Yaskawa INFORM job: A_NAIHAN_0617_1_PAINT_2.JBI

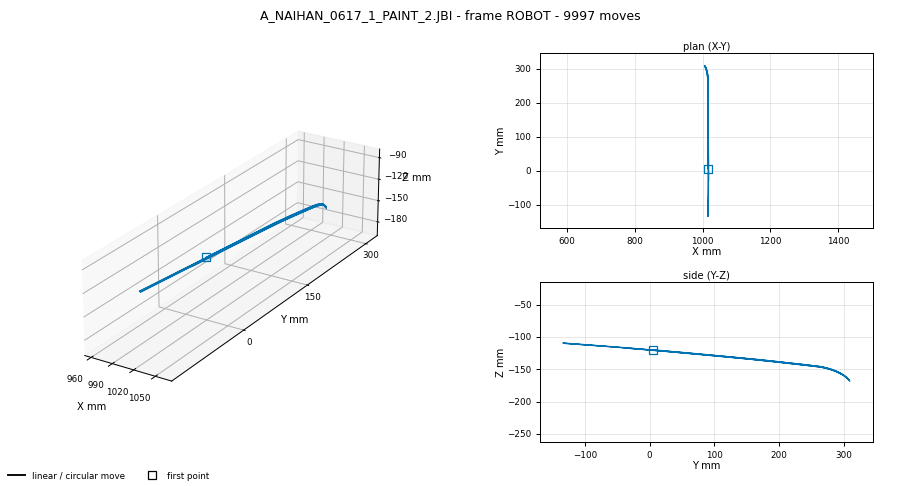
[picture p0: tool path of A_NAIHAN_0617_1_PAINT_2.JBI in frame ROBOT, 9997 of 9997 moves have a stored position in this frame; points joined in program order, loops and branches not executed]
/JOB
//NAME A_NAIHAN_0617_1_PAINT2
//POS
///NPOS 9997,0,0,0,0,0
///TOOL 1
///USER 0
///POSTYPE ROBOT
///RECTAN
///RCONF 0,0,0,0,1,0,0,0,0,0,0,0,0,0,0,0,0,0,0,0,0,0,0,0
C00000=1015.956,5.375,-119.573,-24.182,21.519,-42.790
C00001=1015.955,5.769,-119.606,-24.182,21.518,-42.785
C00002=1015.954,6.162,-119.640,-24.183,21.519,-42.779
C00003=1015.954,6.555,-119.673,-24.184,21.517,-42.775
C00004=1015.952,6.948,-119.706,-24.185,21.517,-42.770
C00005=1015.951,7.339,-119.740,-24.185,21.517,-42.764
C00006=1015.951,7.726,-119.773,-24.186,21.516,-42.761
C00007=1015.950,8.110,-119.806,-24.187,21.516,-42.755
C00008=1015.949,8.491,-119.838,-24.187,21.515,-42.751
C00009=1015.948,8.869,-119.869,-24.188,21.515,-42.746
C00010=1015.947,9.245,-119.902,-24.189,21.514,-42.740
C00011=1015.945,9.621,-119.935,-24.189,21.514,-42.737
C00012=1015.945,9.998,-119.966,-24.190,21.513,-42.731
C00013=1015.944,10.376,-119.999,-24.191,21.513,-42.726
C00014=1015.943,10.757,-120.031,-24.191,21.513,-42.722
C00015=1015.942,11.139,-120.064,-24.192,21.512,-42.716
C00016=1015.940,11.526,-120.098,-24.192,21.511,-42.713
C00017=1015.940,11.912,-120.131,-24.193,21.512,-42.707
C00018=1015.938,12.298,-120.164,-24.193,21.510,-42.703
C00019=1015.938,12.685,-120.197,-24.194,21.510,-42.698
C00020=1015.936,13.071,-120.230,-24.195,21.511,-42.693
C00021=1015.935,13.458,-120.263,-24.196,21.509,-42.689
C00022=1015.933,13.845,-120.297,-24.196,21.509,-42.683
C00023=1015.933,14.233,-120.330,-24.197,21.509,-42.680
C00024=1015.931,14.621,-120.363,-24.198,21.508,-42.674
C00025=1015.930,15.011,-120.397,-24.198,21.508,-42.670
C00026=1015.928,15.400,-120.430,-24.199,21.507,-42.665
C00027=1015.927,15.790,-120.464,-24.200,21.507,-42.659
C00028=1015.927,16.181,-120.498,-24.200,21.506,-42.656
C00029=1015.925,16.573,-120.531,-24.201,21.506,-42.650
C00030=1015.923,16.965,-120.565,-24.201,21.505,-42.646
C00031=1015.922,17.359,-120.599,-24.202,21.505,-42.641
C00032=1015.921,17.753,-120.633,-24.203,21.505,-42.635
C00033=1015.920,18.148,-120.667,-24.203,21.504,-42.632
C00034=1015.917,18.544,-120.701,-24.204,21.503,-42.626
C00035=1015.917,18.940,-120.736,-24.205,21.503,-42.622
C00036=1015.915,19.338,-120.770,-24.205,21.503,-42.617
C00037=1015.914,19.548,-120.788,-24.206,21.503,-42.613
C00038=1015.913,19.785,-120.809,-24.206,21.502,-42.610
C00039=1015.912,20.051,-120.831,-24.207,21.503,-42.606
C00040=1015.912,20.337,-120.857,-24.207,21.501,-42.604
C00041=1015.910,20.635,-120.882,-24.207,21.501,-42.602
C00042=1015.909,20.926,-120.907,-24.208,21.502,-42.599
C00043=1015.908,21.198,-120.931,-24.208,21.501,-42.597
C00044=1015.907,21.443,-120.952,-24.209,21.501,-42.593
C00045=1015.905,21.856,-120.988,-24.210,21.501,-42.586
C00046=1015.904,22.231,-121.020,-24.210,21.500,-42.584
C00047=1015.902,22.553,-121.049,-24.211,21.500,-42.580
C00048=1015.901,22.819,-121.071,-24.211,21.500,-42.577
C00049=1015.900,23.051,-121.092,-24.211,21.499,-42.573
C00050=1015.899,23.286,-121.112,-24.212,21.498,-42.567
C00051=1015.898,23.557,-121.136,-24.213,21.498,-42.564
C00052=1015.897,23.888,-121.165,-24.213,21.498,-42.562
C00053=1015.895,24.271,-121.198,-24.213,21.497,-42.558
C00054=1015.893,24.669,-121.233,-24.214,21.497,-42.553
C00055=1015.891,25.069,-121.267,-24.215,21.497,-42.549
C00056=1015.890,25.468,-121.302,-24.215,21.496,-42.543
C00057=1015.888,25.868,-121.337,-24.216,21.496,-42.540
C00058=1015.886,26.267,-121.372,-24.217,21.496,-42.534
C00059=1015.884,26.666,-121.407,-24.218,21.495,-42.529
C00060=1015.882,27.066,-121.441,-24.218,21.494,-42.525
C00061=1015.881,27.465,-121.476,-24.219,21.495,-42.520
C00062=1015.879,27.865,-121.511,-24.219,21.493,-42.516
C00063=1015.877,28.264,-121.545,-24.220,21.493,-42.510
C00064=1015.875,28.664,-121.581,-24.221,21.493,-42.507
C00065=1015.873,29.063,-121.616,-24.221,21.492,-42.501
C00066=1015.872,29.462,-121.651,-24.222,21.492,-42.497
C00067=1015.869,29.863,-121.686,-24.223,21.492,-42.492
C00068=1015.867,30.262,-121.720,-24.223,21.491,-42.488
C00069=1015.865,30.661,-121.756,-24.224,21.491,-42.483
C00070=1015.863,31.061,-121.790,-24.224,21.490,-42.479
C00071=1015.861,31.461,-121.826,-24.225,21.490,-42.474
C00072=1015.859,31.860,-121.861,-24.226,21.489,-42.469
C00073=1015.857,32.260,-121.895,-24.226,21.489,-42.464
C00074=1015.855,32.659,-121.930,-24.227,21.489,-42.461
C00075=1015.853,33.059,-121.966,-24.228,21.489,-42.455
C00076=1015.850,33.459,-122.001,-24.228,21.487,-42.451
C00077=1015.849,33.858,-122.036,-24.229,21.488,-42.446
C00078=1015.846,34.258,-122.071,-24.229,21.487,-42.442
C00079=1015.844,34.658,-122.106,-24.230,21.486,-42.437
C00080=1015.841,35.057,-122.142,-24.231,21.486,-42.433
C00081=1015.840,35.457,-122.176,-24.231,21.486,-42.428
C00082=1015.837,35.857,-122.211,-24.232,21.486,-42.424
C00083=1015.835,36.256,-122.247,-24.233,21.485,-42.418
C00084=1015.832,36.656,-122.282,-24.233,21.484,-42.414
C00085=1015.830,37.057,-122.317,-24.234,21.485,-42.409
C00086=1015.828,37.456,-122.353,-24.235,21.484,-42.405
C00087=1015.825,37.856,-122.388,-24.235,21.483,-42.400
C00088=1015.823,38.256,-122.423,-24.236,21.483,-42.396
C00089=1015.821,38.655,-122.459,-24.237,21.483,-42.391
C00090=1015.818,39.056,-122.494,-24.237,21.483,-42.387
C00091=1015.816,39.455,-122.529,-24.238,21.482,-42.383
C00092=1015.813,39.855,-122.565,-24.238,21.481,-42.378
C00093=1015.811,40.256,-122.600,-24.239,21.481,-42.374
C00094=1015.809,40.655,-122.635,-24.240,21.481,-42.369
C00095=1015.806,41.055,-122.670,-24.240,21.481,-42.365
C00096=1015.804,41.455,-122.706,-24.241,21.480,-42.359
C00097=1015.801,41.855,-122.742,-24.241,21.479,-42.356
C00098=1015.798,42.255,-122.777,-24.242,21.479,-42.352
C00099=1015.796,42.654,-122.812,-24.243,21.479,-42.347
C00100=1015.794,43.055,-122.847,-24.243,21.479,-42.343
C00101=1015.791,43.455,-122.884,-24.244,21.479,-42.338
C00102=1015.788,43.855,-122.918,-24.244,21.477,-42.333
C00103=1015.786,44.255,-122.954,-24.245,21.477,-42.330
C00104=1015.783,44.655,-122.990,-24.246,21.477,-42.325
C00105=1015.780,45.055,-123.025,-24.246,21.477,-42.321
C00106=1015.778,45.455,-123.061,-24.247,21.477,-42.316
C00107=1015.775,45.855,-123.096,-24.247,21.475,-42.311
C00108=1015.772,46.255,-123.132,-24.248,21.475,-42.308
C00109=1015.770,46.655,-123.168,-24.249,21.475,-42.302
C00110=1015.766,47.055,-123.203,-24.249,21.475,-42.299
C00111=1015.764,47.455,-123.239,-24.250,21.474,-42.295
C00112=1015.761,47.855,-123.274,-24.251,21.474,-42.290
C00113=1015.758,48.256,-123.311,-24.251,21.474,-42.286
C00114=1015.756,48.656,-123.345,-24.251,21.472,-42.282
C00115=1015.753,49.056,-123.381,-24.252,21.473,-42.277
C00116=1015.750,49.455,-123.417,-24.253,21.472,-42.273
C00117=1015.747,49.856,-123.452,-24.254,21.472,-42.268
C00118=1015.744,50.256,-123.489,-24.254,21.472,-42.264
C00119=1015.740,50.656,-123.524,-24.255,21.471,-42.260
C00120=1015.739,51.056,-123.560,-24.255,21.471,-42.255
C00121=1015.735,51.457,-123.595,-24.256,21.471,-42.251
C00122=1015.732,51.857,-123.631,-24.256,21.470,-42.247
C00123=1015.729,52.257,-123.667,-24.257,21.469,-42.243
C00124=1015.726,52.657,-123.703,-24.258,21.469,-42.238
C00125=1015.723,53.057,-123.739,-24.258,21.469,-42.234
C00126=1015.719,53.457,-123.774,-24.259,21.468,-42.230
C00127=1015.717,53.857,-123.810,-24.259,21.468,-42.225
C00128=1015.714,54.257,-123.846,-24.260,21.468,-42.221
C00129=1015.711,54.658,-123.882,-24.260,21.468,-42.218
C00130=1015.708,55.058,-123.918,-24.261,21.468,-42.212
C00131=1015.705,55.458,-123.953,-24.262,21.467,-42.209
C00132=1015.702,55.858,-123.989,-24.262,21.467,-42.205
C00133=1015.698,56.258,-124.026,-24.263,21.465,-42.201
C00134=1015.695,56.659,-124.062,-24.264,21.466,-42.196
C00135=1015.691,57.059,-124.098,-24.264,21.465,-42.192
C00136=1015.688,57.459,-124.133,-24.264,21.465,-42.188
C00137=1015.685,57.859,-124.169,-24.265,21.465,-42.183
C00138=1015.682,58.259,-124.205,-24.266,21.464,-42.179
C00139=1015.679,58.659,-124.241,-24.266,21.464,-42.175
C00140=1015.675,59.059,-124.277,-24.267,21.463,-42.172
C00141=1015.671,59.460,-124.313,-24.268,21.464,-42.166
C00142=1015.668,59.860,-124.349,-24.268,21.463,-42.163
C00143=1015.665,60.260,-124.385,-24.269,21.463,-42.159
C00144=1015.661,60.660,-124.421,-24.269,21.462,-42.155
C00145=1015.658,61.060,-124.457,-24.270,21.462,-42.150
C00146=1015.655,61.460,-124.493,-24.270,21.462,-42.146
C00147=1015.651,61.861,-124.529,-24.271,21.461,-42.142
C00148=1015.648,62.261,-124.565,-24.271,21.461,-42.139
C00149=1015.644,62.681,-124.603,-24.272,21.460,-42.133
C00150=1015.642,62.934,-124.626,-24.272,21.460,-42.131
C00151=1015.640,63.201,-124.650,-24.273,21.460,-42.129
C00152=1015.638,63.450,-124.673,-24.273,21.459,-42.127
C00153=1015.636,63.668,-124.693,-24.274,21.460,-42.124
C00154=1015.634,63.875,-124.711,-24.274,21.460,-42.122
C00155=1015.631,64.093,-124.730,-24.274,21.459,-42.120
C00156=1015.629,64.322,-124.751,-24.274,21.459,-42.116
C00157=1015.627,64.558,-124.773,-24.275,21.459,-42.115
C00158=1015.625,64.794,-124.794,-24.275,21.458,-42.113
C00159=1015.623,65.024,-124.815,-24.275,21.458,-42.111
C00160=1015.621,65.245,-124.835,-24.276,21.459,-42.108
C00161=1015.619,65.458,-124.853,-24.276,21.458,-42.106
C00162=1015.616,65.866,-124.891,-24.277,21.458,-42.102
C00163=1015.611,66.264,-124.927,-24.277,21.457,-42.098
C00164=1015.609,66.665,-124.963,-24.278,21.457,-42.094
C00165=1015.604,67.067,-124.999,-24.278,21.457,-42.089
C00166=1015.600,67.470,-125.036,-24.279,21.457,-42.085
C00167=1015.597,67.875,-125.072,-24.279,21.456,-42.082
C00168=1015.593,68.281,-125.110,-24.280,21.456,-42.078
C00169=1015.590,68.689,-125.146,-24.280,21.455,-42.074
C00170=1015.586,69.097,-125.183,-24.281,21.455,-42.069
C00171=1015.581,69.507,-125.221,-24.282,21.455,-42.065
C00172=1015.577,69.918,-125.258,-24.282,21.454,-42.061
C00173=1015.573,70.330,-125.295,-24.283,21.454,-42.058
C00174=1015.570,70.741,-125.332,-24.283,21.453,-42.054
C00175=1015.566,71.152,-125.369,-24.284,21.454,-42.049
C00176=1015.562,71.563,-125.406,-24.285,21.453,-42.045
C00177=1015.557,71.975,-125.444,-24.285,21.453,-42.041
C00178=1015.553,72.388,-125.482,-24.285,21.452,-42.037
C00179=1015.550,72.804,-125.520,-24.286,21.452,-42.034
C00180=1015.545,73.221,-125.557,-24.287,21.452,-42.028
C00181=1015.541,73.641,-125.596,-24.287,21.452,-42.025
C00182=1015.539,73.853,-125.615,-24.288,21.451,-42.023
C00183=1015.537,74.065,-125.634,-24.288,21.451,-42.021
C00184=1015.535,74.278,-125.653,-24.288,21.451,-42.019
C00185=1015.532,74.490,-125.673,-24.288,21.451,-42.017
C00186=1015.530,74.704,-125.692,-24.289,21.450,-42.015
C00187=1015.528,74.918,-125.712,-24.289,21.451,-42.012
C00188=1015.526,75.131,-125.731,-24.289,21.451,-42.010
C00189=1015.523,75.344,-125.751,-24.290,21.450,-42.008
C00190=1015.519,75.763,-125.789,-24.290,21.450,-42.004
C00191=1015.514,76.175,-125.826,-24.291,21.449,-42.001
C00192=1015.511,76.577,-125.862,-24.291,21.449,-41.997
C00193=1015.507,76.972,-125.898,-24.292,21.449,-41.994
C00194=1015.503,77.360,-125.934,-24.292,21.448,-41.989
C00195=1015.498,77.746,-125.969,-24.293,21.447,-41.986
C00196=1015.495,78.133,-126.005,-24.293,21.448,-41.980
C00197=1015.490,78.523,-126.040,-24.294,21.447,-41.977
C00198=1015.485,78.920,-126.076,-24.294,21.447,-41.973
C00199=1015.481,79.326,-126.113,-24.295,21.447,-41.970
C00200=1015.477,79.740,-126.152,-24.296,21.447,-41.966
C00201=1015.475,79.950,-126.170,-24.296,21.446,-41.964
C00202=1015.473,80.162,-126.190,-24.296,21.446,-41.962
C00203=1015.471,80.375,-126.209,-24.296,21.446,-41.960
C00204=1015.468,80.588,-126.228,-24.297,21.446,-41.958
C00205=1015.466,80.800,-126.247,-24.297,21.445,-41.956
C00206=1015.463,81.013,-126.267,-24.297,21.445,-41.955
C00207=1015.461,81.225,-126.287,-24.297,21.445,-41.953
C00208=1015.459,81.437,-126.306,-24.298,21.445,-41.951
C00209=1015.456,81.650,-126.326,-24.298,21.445,-41.949
C00210=1015.453,81.862,-126.345,-24.298,21.444,-41.947
C00211=1015.451,82.073,-126.364,-24.299,21.445,-41.944
C00212=1015.449,82.284,-126.384,-24.299,21.444,-41.942
C00213=1015.444,82.705,-126.422,-24.299,21.444,-41.938
C00214=1015.440,83.126,-126.460,-24.300,21.444,-41.935
C00215=1015.434,83.545,-126.499,-24.300,21.444,-41.931
C00216=1015.430,83.962,-126.537,-24.301,21.443,-41.927
C00217=1015.425,84.378,-126.575,-24.301,21.443,-41.923
C00218=1015.420,84.792,-126.613,-24.302,21.443,-41.920
C00219=1015.416,85.204,-126.651,-24.302,21.442,-41.916
C00220=1015.411,85.615,-126.688,-24.303,21.442,-41.912
C00221=1015.407,86.024,-126.725,-24.303,21.441,-41.908
C00222=1015.401,86.431,-126.763,-24.304,21.442,-41.905
C00223=1015.397,86.837,-126.800,-24.304,21.441,-41.901
C00224=1015.392,87.240,-126.836,-24.305,21.441,-41.898
C00225=1015.388,87.636,-126.873,-24.305,21.440,-41.894
C00226=1015.383,88.023,-126.908,-24.306,21.440,-41.890
C00227=1015.378,88.407,-126.944,-24.307,21.440,-41.887
C00228=1015.374,88.790,-126.979,-24.307,21.440,-41.883
C00229=1015.369,89.176,-127.014,-24.308,21.439,-41.879
C00230=1015.364,89.569,-127.050,-24.308,21.439,-41.875
C00231=1015.360,89.967,-127.087,-24.309,21.439,-41.872
C00232=1015.355,90.367,-127.124,-24.309,21.439,-41.868
C00233=1015.350,90.766,-127.160,-24.310,21.438,-41.865
C00234=1015.344,91.165,-127.197,-24.310,21.438,-41.861
C00235=1015.340,91.563,-127.234,-24.311,21.438,-41.857
C00236=1015.335,91.963,-127.271,-24.311,21.438,-41.854
C00237=1015.330,92.362,-127.307,-24.312,21.437,-41.850
C00238=1015.325,92.761,-127.344,-24.312,21.437,-41.846
C00239=1015.320,93.160,-127.380,-24.312,21.437,-41.844
C00240=1015.315,93.559,-127.416,-24.313,21.436,-41.841
C00241=1015.310,93.958,-127.453,-24.313,21.436,-41.837
C00242=1015.304,94.357,-127.490,-24.314,21.435,-41.833
C00243=1015.300,94.756,-127.527,-24.315,21.436,-41.830
C00244=1015.294,95.155,-127.564,-24.315,21.435,-41.826
C00245=1015.289,95.553,-127.600,-24.316,21.435,-41.822
C00246=1015.284,95.952,-127.637,-24.316,21.435,-41.819
C00247=1015.279,96.351,-127.674,-24.317,21.435,-41.815
C00248=1015.274,96.750,-127.710,-24.317,21.434,-41.811
C00249=1015.268,97.149,-127.747,-24.318,21.434,-41.808
C00250=1015.263,97.547,-127.783,-24.318,21.433,-41.806
C00251=1015.258,97.947,-127.820,-24.318,21.433,-41.802
C00252=1015.253,98.346,-127.858,-24.319,21.432,-41.798
C00253=1015.248,98.744,-127.894,-24.319,21.433,-41.795
C00254=1015.242,99.143,-127.931,-24.320,21.432,-41.791
C00255=1015.237,99.542,-127.968,-24.320,21.432,-41.787
C00256=1015.232,99.941,-128.004,-24.321,21.432,-41.784
C00257=1015.226,100.339,-128.041,-24.322,21.432,-41.780
C00258=1015.220,100.738,-128.077,-24.322,21.431,-41.778
C00259=1015.215,101.137,-128.115,-24.322,21.431,-41.775
C00260=1015.210,101.535,-128.151,-24.323,21.431,-41.771
C00261=1015.204,101.934,-128.188,-24.323,21.430,-41.767
C00262=1015.199,102.333,-128.225,-24.324,21.430,-41.763
C00263=1015.193,102.731,-128.262,-24.324,21.430,-41.760
C00264=1015.188,103.130,-128.298,-24.325,21.430,-41.756
C00265=1015.182,103.528,-128.335,-24.325,21.430,-41.754
C00266=1015.176,103.927,-128.372,-24.326,21.429,-41.751
C00267=1015.171,104.326,-128.408,-24.326,21.429,-41.747
C00268=1015.165,104.724,-128.445,-24.327,21.429,-41.743
C00269=1015.160,105.123,-128.482,-24.327,21.429,-41.740
C00270=1015.154,105.521,-128.519,-24.328,21.428,-41.736
C00271=1015.148,105.920,-128.555,-24.328,21.428,-41.734
C00272=1015.142,106.318,-128.593,-24.328,21.427,-41.730
C00273=1015.137,106.718,-128.629,-24.329,21.427,-41.727
C00274=1015.131,107.115,-128.666,-24.330,21.427,-41.723
C00275=1015.125,107.514,-128.703,-24.330,21.427,-41.719
C00276=1015.119,107.913,-128.740,-24.330,21.426,-41.717
C00277=1015.113,108.311,-128.776,-24.331,21.426,-41.714
C00278=1015.108,108.709,-128.813,-24.331,21.426,-41.710
C00279=1015.102,109.109,-128.850,-24.332,21.426,-41.707
C00280=1015.096,109.506,-128.887,-24.332,21.426,-41.703
C00281=1015.089,109.906,-128.924,-24.333,21.425,-41.701
C00282=1015.083,110.303,-128.961,-24.333,21.425,-41.697
C00283=1015.078,110.702,-128.998,-24.334,21.425,-41.694
C00284=1015.072,111.100,-129.035,-24.334,21.425,-41.690
C00285=1015.066,111.499,-129.071,-24.334,21.424,-41.688
C00286=1015.062,111.764,-129.095,-24.335,21.424,-41.685
C00287=1015.058,112.030,-129.121,-24.335,21.424,-41.683
C00288=1015.053,112.296,-129.145,-24.335,21.424,-41.681
C00289=1015.047,112.694,-129.182,-24.336,21.423,-41.677
C00290=1015.042,113.093,-129.219,-24.336,21.423,-41.675
C00291=1015.036,113.491,-129.256,-24.337,21.423,-41.671
C00292=1015.029,113.890,-129.293,-24.337,21.422,-41.668
C00293=1015.023,114.288,-129.330,-24.338,21.423,-41.664
C00294=1015.017,114.686,-129.366,-24.338,21.422,-41.662
C00295=1015.010,115.086,-129.403,-24.339,21.422,-41.659
C00296=1015.004,115.483,-129.440,-24.339,21.422,-41.655
C00297=1014.998,115.883,-129.477,-24.340,21.422,-41.652
C00298=1014.992,116.280,-129.514,-24.340,21.421,-41.649
C00299=1014.985,116.679,-129.550,-24.340,21.420,-41.646
C00300=1014.979,117.077,-129.588,-24.341,21.421,-41.642
C00301=1014.973,117.476,-129.624,-24.341,21.420,-41.638
C00302=1014.966,117.874,-129.662,-24.342,21.420,-41.637
C00303=1014.960,118.272,-129.698,-24.342,21.420,-41.633
C00304=1014.953,118.671,-129.735,-24.343,21.420,-41.629
C00305=1014.947,119.069,-129.772,-24.343,21.420,-41.626
C00306=1014.940,119.468,-129.809,-24.343,21.419,-41.624
C00307=1014.934,119.866,-129.846,-24.344,21.419,-41.620
C00308=1014.927,120.264,-129.883,-24.345,21.419,-41.617
C00309=1014.921,120.663,-129.921,-24.345,21.418,-41.614
C00310=1014.914,121.061,-129.957,-24.345,21.418,-41.611
C00311=1014.908,121.460,-129.995,-24.346,21.418,-41.607
C00312=1014.902,121.858,-130.032,-24.346,21.417,-41.605
C00313=1014.896,122.257,-130.069,-24.347,21.418,-41.602
C00314=1014.890,122.655,-130.106,-24.347,21.417,-41.598
C00315=1014.884,123.054,-130.144,-24.348,21.418,-41.595
C00316=1014.878,123.451,-130.181,-24.348,21.416,-41.592
C00317=1014.871,123.851,-130.218,-24.348,21.417,-41.589
C00318=1014.864,124.249,-130.255,-24.349,21.416,-41.585
C00319=1014.859,124.647,-130.293,-24.349,21.416,-41.583
C00320=1014.852,125.046,-130.329,-24.350,21.416,-41.580
C00321=1014.846,125.445,-130.367,-24.350,21.416,-41.576
C00322=1014.840,125.842,-130.404,-24.350,21.415,-41.574
C00323=1014.832,126.241,-130.441,-24.351,21.415,-41.571
C00324=1014.826,126.640,-130.479,-24.351,21.415,-41.567
C00325=1014.819,127.038,-130.516,-24.352,21.415,-41.565
C00326=1014.814,127.437,-130.553,-24.352,21.414,-41.561
C00327=1014.807,127.835,-130.591,-24.353,21.415,-41.558
C00328=1014.800,128.234,-130.627,-24.353,21.414,-41.555
C00329=1014.794,128.632,-130.665,-24.354,21.414,-41.552
C00330=1014.787,129.031,-130.702,-24.354,21.413,-41.550
C00331=1014.780,129.429,-130.740,-24.354,21.413,-41.547
C00332=1014.773,129.828,-130.777,-24.355,21.413,-41.543
C00333=1014.767,130.226,-130.814,-24.355,21.413,-41.541
C00334=1014.761,130.624,-130.851,-24.356,21.413,-41.538
C00335=1014.754,131.023,-130.888,-24.356,21.413,-41.534
C00336=1014.747,131.421,-130.926,-24.356,21.412,-41.532
C00337=1014.740,131.820,-130.963,-24.357,21.412,-41.528
C00338=1014.733,132.219,-131.001,-24.357,21.412,-41.525
C00339=1014.726,132.618,-131.038,-24.358,21.411,-41.523
C00340=1014.720,133.016,-131.075,-24.358,21.412,-41.519
C00341=1014.712,133.415,-131.112,-24.358,21.411,-41.517
C00342=1014.706,133.814,-131.149,-24.359,21.411,-41.514
C00343=1014.699,134.212,-131.187,-24.359,21.411,-41.510
C00344=1014.692,134.611,-131.224,-24.360,21.410,-41.508
C00345=1014.685,135.009,-131.262,-24.360,21.411,-41.505
C00346=1014.678,135.404,-131.298,-24.360,21.410,-41.502
C00347=1014.672,135.776,-131.333,-24.361,21.409,-41.500
C00348=1014.666,136.115,-131.365,-24.361,21.410,-41.497
C00349=1014.660,136.433,-131.395,-24.361,21.409,-41.495
C00350=1014.654,136.749,-131.425,-24.362,21.409,-41.491
C00351=1014.648,137.085,-131.456,-24.363,21.410,-41.488
C00352=1014.641,137.455,-131.490,-24.363,21.408,-41.486
C00353=1014.635,137.856,-131.527,-24.363,21.408,-41.484
C00354=1014.630,138.062,-131.547,-24.363,21.408,-41.482
C00355=1014.627,138.279,-131.568,-24.364,21.408,-41.480
C00356=1014.623,138.516,-131.590,-24.364,21.408,-41.478
C00357=1014.618,138.775,-131.614,-24.364,21.407,-41.476
C00358=1014.612,139.054,-131.639,-24.364,21.408,-41.475
C00359=1014.608,139.341,-131.667,-24.365,21.408,-41.473
C00360=1014.602,139.629,-131.694,-24.365,21.408,-41.471
C00361=1014.597,139.906,-131.720,-24.365,21.408,-41.470
C00362=1014.592,140.164,-131.744,-24.366,21.408,-41.468
C00363=1014.588,140.400,-131.766,-24.366,21.408,-41.466
C00364=1014.581,140.817,-131.805,-24.366,21.407,-41.462
C00365=1014.573,141.222,-131.843,-24.366,21.406,-41.460
C00366=1014.565,141.627,-131.881,-24.367,21.407,-41.457
C00367=1014.558,142.033,-131.918,-24.368,21.406,-41.453
C00368=1014.550,142.440,-131.957,-24.368,21.406,-41.451
C00369=1014.543,142.848,-131.995,-24.368,21.406,-41.448
C00370=1014.534,143.257,-132.033,-24.369,21.405,-41.445
C00371=1014.527,143.666,-132.072,-24.369,21.406,-41.442
C00372=1014.519,144.076,-132.110,-24.370,21.405,-41.438
C00373=1014.511,144.487,-132.149,-24.370,21.405,-41.436
C00374=1014.503,144.898,-132.187,-24.370,21.405,-41.432
C00375=1014.495,145.311,-132.226,-24.371,21.404,-41.431
C00376=1014.487,145.723,-132.265,-24.371,21.405,-41.427
C00377=1014.479,146.135,-132.303,-24.372,21.404,-41.424
C00378=1014.471,146.548,-132.341,-24.372,21.404,-41.422
C00379=1014.463,146.962,-132.380,-24.372,21.404,-41.418
C00380=1014.455,147.375,-132.418,-24.373,21.403,-41.416
C00381=1014.447,147.789,-132.457,-24.373,21.403,-41.412
C00382=1014.438,148.203,-132.496,-24.374,21.403,-41.409
C00383=1014.431,148.617,-132.535,-24.374,21.403,-41.407
C00384=1014.422,149.030,-132.573,-24.375,21.403,-41.403
C00385=1014.414,149.444,-132.612,-24.375,21.402,-41.401
C00386=1014.405,149.858,-132.651,-24.375,21.402,-41.398
C00387=1014.397,150.273,-132.689,-24.376,21.402,-41.394
C00388=1014.388,150.686,-132.728,-24.376,21.401,-41.392
C00389=1014.381,151.099,-132.767,-24.377,21.402,-41.389
C00390=1014.372,151.513,-132.805,-24.377,21.402,-41.387
C00391=1014.363,151.926,-132.844,-24.377,21.401,-41.383
C00392=1014.355,152.338,-132.882,-24.378,21.401,-41.381
C00393=1014.347,152.750,-132.921,-24.378,21.400,-41.377
C00394=1014.338,153.162,-132.959,-24.378,21.400,-41.375
C00395=1014.329,153.572,-132.997,-24.379,21.401,-41.372
C00396=1014.321,153.983,-133.035,-24.380,21.400,-41.368
C00397=1014.312,154.393,-133.075,-24.380,21.400,-41.366
C00398=1014.304,154.802,-133.113,-24.380,21.400,-41.363
C00399=1014.295,155.211,-133.151,-24.381,21.399,-41.361
C00400=1014.286,155.618,-133.189,-24.381,21.400,-41.358
C00401=1014.278,156.024,-133.227,-24.381,21.399,-41.355
C00402=1014.269,156.430,-133.264,-24.382,21.399,-41.352
C00403=1014.260,156.835,-133.303,-24.382,21.399,-41.350
C00404=1014.252,157.239,-133.340,-24.383,21.398,-41.346
C00405=1014.244,157.642,-133.378,-24.383,21.398,-41.344
C00406=1014.234,158.045,-133.415,-24.383,21.399,-41.341
C00407=1014.225,158.447,-133.453,-24.384,21.397,-41.339
C00408=1014.217,158.847,-133.490,-24.384,21.398,-41.335
C00409=1014.208,159.249,-133.527,-24.384,21.398,-41.333
C00410=1014.199,159.647,-133.565,-24.385,21.397,-41.330
C00411=1014.195,160.045,-133.605,-24.385,21.397,-41.328
C00412=1014.192,160.450,-133.647,-24.386,21.397,-41.325
C00413=1014.192,160.663,-133.669,-24.386,21.397,-41.324
C00414=1014.192,160.887,-133.692,-24.386,21.396,-41.322
C00415=1014.190,161.125,-133.717,-24.386,21.396,-41.320
C00416=1014.190,161.376,-133.743,-24.387,21.397,-41.319
C00417=1014.188,161.638,-133.771,-24.387,21.397,-41.317
C00418=1014.187,161.908,-133.798,-24.387,21.396,-41.315
C00419=1014.186,162.179,-133.827,-24.387,21.396,-41.313
C00420=1014.184,162.448,-133.855,-24.388,21.396,-41.311
C00421=1014.184,162.711,-133.883,-24.388,21.396,-41.309
C00422=1014.182,162.964,-133.909,-24.388,21.395,-41.308
C00423=1014.181,163.200,-133.933,-24.388,21.396,-41.306
C00424=1014.180,163.612,-133.976,-24.389,21.395,-41.304
C00425=1014.179,163.802,-133.997,-24.389,21.395,-41.302
C00426=1014.177,164.188,-134.037,-24.389,21.395,-41.300
C00427=1014.176,164.588,-134.079,-24.390,21.395,-41.297
C00428=1014.174,164.988,-134.121,-24.390,21.395,-41.295
C00429=1014.173,165.389,-134.163,-24.390,21.394,-41.291
C00430=1014.171,165.789,-134.205,-24.391,21.394,-41.289
C00431=1014.169,166.190,-134.248,-24.391,21.395,-41.286
C00432=1014.168,166.590,-134.289,-24.391,21.393,-41.284
C00433=1014.166,166.990,-134.331,-24.392,21.394,-41.280
C00434=1014.165,167.390,-134.373,-24.392,21.394,-41.278
C00435=1014.163,167.791,-134.415,-24.393,21.394,-41.275
C00436=1014.161,168.191,-134.458,-24.393,21.393,-41.273
C00437=1014.160,168.591,-134.499,-24.393,21.393,-41.271
C00438=1014.158,168.993,-134.541,-24.394,21.393,-41.267
C00439=1014.156,169.392,-134.584,-24.394,21.392,-41.265
C00440=1014.155,169.793,-134.626,-24.395,21.392,-41.262
C00441=1014.153,170.193,-134.668,-24.395,21.392,-41.260
C00442=1014.152,170.594,-134.710,-24.395,21.392,-41.256
C00443=1014.150,170.995,-134.753,-24.396,21.392,-41.254
C00444=1014.149,171.395,-134.795,-24.396,21.392,-41.251
C00445=1014.147,171.796,-134.837,-24.396,21.392,-41.249
C00446=1014.146,172.196,-134.880,-24.397,21.391,-41.247
C00447=1014.143,172.597,-134.922,-24.397,21.391,-41.243
C00448=1014.142,172.998,-134.964,-24.397,21.391,-41.242
C00449=1014.141,173.398,-135.006,-24.398,21.390,-41.238
C00450=1014.140,173.799,-135.048,-24.398,21.390,-41.236
C00451=1014.138,174.200,-135.091,-24.399,21.391,-41.233
C00452=1014.136,174.600,-135.133,-24.399,21.390,-41.231
C00453=1014.135,175.001,-135.176,-24.400,21.390,-41.227
C00454=1014.133,175.402,-135.218,-24.400,21.390,-41.225
C00455=1014.132,175.802,-135.261,-24.400,21.390,-41.223
C00456=1014.130,176.203,-135.304,-24.401,21.389,-41.219
C00457=1014.129,176.604,-135.346,-24.401,21.389,-41.218
C00458=1014.128,177.005,-135.388,-24.401,21.389,-41.214
C00459=1014.126,177.405,-135.431,-24.402,21.389,-41.212
C00460=1014.125,177.806,-135.473,-24.402,21.389,-41.209
C00461=1014.123,178.207,-135.516,-24.402,21.388,-41.207
C00462=1014.122,178.608,-135.559,-24.403,21.388,-41.205
C00463=1014.120,179.009,-135.602,-24.403,21.388,-41.201
C00464=1014.119,179.410,-135.644,-24.403,21.388,-41.199
C00465=1014.117,179.810,-135.687,-24.404,21.388,-41.196
C00466=1014.116,180.211,-135.730,-24.404,21.388,-41.194
C00467=1014.114,180.612,-135.772,-24.405,21.387,-41.190
C00468=1014.113,181.012,-135.815,-24.405,21.387,-41.188
C00469=1014.111,181.413,-135.857,-24.405,21.387,-41.186
C00470=1014.110,181.814,-135.900,-24.406,21.387,-41.183
C00471=1014.109,182.215,-135.943,-24.406,21.386,-41.181
C00472=1014.108,182.616,-135.986,-24.407,21.387,-41.177
C00473=1014.105,183.017,-136.029,-24.407,21.386,-41.176
C00474=1014.104,183.418,-136.072,-24.407,21.386,-41.172
C00475=1014.103,183.819,-136.115,-24.408,21.386,-41.170
C00476=1014.102,184.220,-136.158,-24.408,21.386,-41.168
C00477=1014.100,184.620,-136.201,-24.409,21.386,-41.165
C00478=1014.100,185.022,-136.244,-24.409,21.385,-41.162
C00479=1014.098,185.423,-136.286,-24.409,21.385,-41.159
C00480=1014.097,185.823,-136.329,-24.410,21.385,-41.157
C00481=1014.095,186.225,-136.373,-24.410,21.384,-41.155
C00482=1014.093,186.626,-136.415,-24.410,21.384,-41.151
C00483=1014.092,187.026,-136.458,-24.411,21.384,-41.150
C00484=1014.091,187.428,-136.501,-24.411,21.385,-41.146
C00485=1014.090,187.828,-136.544,-24.411,21.384,-41.144
C00486=1014.089,188.229,-136.588,-24.412,21.384,-41.141
C00487=1014.087,188.631,-136.631,-24.412,21.384,-41.139
C00488=1014.086,189.032,-136.674,-24.412,21.384,-41.137
C00489=1014.085,189.433,-136.717,-24.413,21.383,-41.133
C00490=1014.084,189.834,-136.760,-24.413,21.383,-41.131
C00491=1014.082,190.235,-136.804,-24.414,21.383,-41.128
C00492=1014.081,190.636,-136.847,-24.414,21.383,-41.126
C00493=1014.080,191.037,-136.890,-24.414,21.382,-41.124
C00494=1014.079,191.438,-136.933,-24.415,21.382,-41.120
C00495=1014.078,191.839,-136.977,-24.415,21.382,-41.118
C00496=1014.077,192.240,-137.020,-24.415,21.382,-41.115
C00497=1014.076,192.641,-137.063,-24.416,21.382,-41.113
C00498=1014.075,193.042,-137.107,-24.416,21.382,-41.109
C00499=1014.073,193.443,-137.150,-24.417,21.382,-41.108
C00500=1014.072,193.844,-137.194,-24.417,21.381,-41.105
C00501=1014.071,194.245,-137.237,-24.417,21.381,-41.102
C00502=1014.070,194.647,-137.281,-24.418,21.381,-41.100
C00503=1014.068,195.047,-137.324,-24.418,21.381,-41.097
C00504=1014.068,195.449,-137.367,-24.418,21.380,-41.094
C00505=1014.066,195.850,-137.411,-24.419,21.381,-41.091
C00506=1014.065,196.251,-137.454,-24.419,21.380,-41.089
C00507=1014.065,196.653,-137.498,-24.419,21.380,-41.087
C00508=1014.063,197.054,-137.542,-24.420,21.380,-41.084
C00509=1014.062,197.455,-137.584,-24.420,21.380,-41.082
C00510=1014.061,197.855,-137.628,-24.421,21.380,-41.078
C00511=1014.060,198.257,-137.672,-24.421,21.379,-41.076
C00512=1014.059,198.658,-137.716,-24.421,21.379,-41.074
C00513=1014.059,199.056,-137.759,-24.422,21.379,-41.071
C00514=1014.057,199.445,-137.802,-24.422,21.379,-41.069
C00515=1014.056,199.846,-137.845,-24.423,21.378,-41.065
C00516=1014.055,200.059,-137.868,-24.423,21.378,-41.065
C00517=1014.055,200.281,-137.893,-24.423,21.378,-41.063
C00518=1014.055,200.510,-137.918,-24.423,21.378,-41.061
C00519=1014.054,200.737,-137.942,-24.423,21.379,-41.060
C00520=1014.053,201.145,-137.987,-24.424,21.378,-41.058
C00521=1014.053,201.497,-138.025,-24.424,21.378,-41.054
C00522=1014.052,201.846,-138.063,-24.424,21.378,-41.052
C00523=1014.051,202.233,-138.107,-24.425,21.378,-41.051
C00524=1014.055,203.448,-138.241,-24.373,21.403,-41.416
C00525=1014.057,203.697,-138.268,-24.373,21.404,-41.415
C00526=1014.059,203.946,-138.296,-24.373,21.403,-41.414
C00527=1014.061,204.194,-138.323,-24.373,21.403,-41.412
C00528=1014.063,204.443,-138.350,-24.374,21.404,-41.411
C00529=1014.064,204.691,-138.377,-24.373,21.403,-41.410
C00530=1014.066,204.940,-138.404,-24.374,21.403,-41.409
C00531=1014.067,205.188,-138.432,-24.374,21.403,-41.407
C00532=1014.069,205.437,-138.459,-24.374,21.402,-41.407
C00533=1014.071,205.685,-138.487,-24.374,21.403,-41.405
C00534=1014.073,205.933,-138.514,-24.375,21.403,-41.403
C00535=1014.074,206.182,-138.541,-24.375,21.402,-41.401
C00536=1014.076,206.431,-138.568,-24.375,21.402,-41.401
C00537=1014.077,206.679,-138.596,-24.375,21.402,-41.399
C00538=1014.080,206.927,-138.624,-24.375,21.402,-41.398
C00539=1014.081,207.176,-138.651,-24.375,21.402,-41.398
C00540=1014.083,207.425,-138.678,-24.376,21.402,-41.396
C00541=1014.085,207.673,-138.705,-24.376,21.402,-41.394
C00542=1014.086,207.922,-138.733,-24.376,21.402,-41.392
C00543=1014.088,208.164,-138.760,-24.376,21.401,-41.392
C00544=1014.090,208.407,-138.786,-24.376,21.402,-41.391
C00545=1014.091,208.649,-138.814,-24.377,21.402,-41.389
C00546=1014.093,208.892,-138.840,-24.377,21.401,-41.388
C00547=1014.095,209.134,-138.867,-24.377,21.402,-41.387
C00548=1014.097,209.377,-138.893,-24.377,21.401,-41.385
C00549=1014.099,209.620,-138.921,-24.377,21.401,-41.383
C00550=1014.100,209.862,-138.947,-24.377,21.401,-41.383
C00551=1014.102,210.110,-138.975,-24.378,21.401,-41.381
C00552=1014.104,210.359,-139.003,-24.378,21.401,-41.379
C00553=1014.106,210.608,-139.030,-24.378,21.401,-41.378
C00554=1014.107,210.856,-139.058,-24.378,21.400,-41.377
C00555=1014.110,211.104,-139.085,-24.378,21.400,-41.375
C00556=1014.111,211.353,-139.112,-24.379,21.401,-41.374
C00557=1014.113,211.601,-139.140,-24.379,21.401,-41.372
C00558=1014.115,211.850,-139.167,-24.379,21.400,-41.372
C00559=1014.117,212.099,-139.195,-24.379,21.400,-41.370
C00560=1014.119,212.347,-139.223,-24.380,21.400,-41.368
C00561=1014.121,212.596,-139.250,-24.380,21.400,-41.366
C00562=1014.123,212.844,-139.278,-24.380,21.400,-41.366
C00563=1014.124,213.092,-139.306,-24.380,21.400,-41.365
C00564=1014.127,213.340,-139.333,-24.380,21.400,-41.363
C00565=1014.128,213.589,-139.361,-24.381,21.400,-41.361
C00566=1014.130,213.838,-139.388,-24.381,21.400,-41.359
C00567=1014.132,214.086,-139.416,-24.381,21.399,-41.359
C00568=1014.134,214.335,-139.443,-24.381,21.399,-41.357
C00569=1014.137,214.583,-139.471,-24.381,21.400,-41.356
C00570=1014.138,214.832,-139.499,-24.382,21.399,-41.354
C00571=1014.141,215.074,-139.526,-24.382,21.398,-41.353
C00572=1014.142,215.316,-139.553,-24.382,21.399,-41.352
C00573=1014.144,215.560,-139.580,-24.382,21.399,-41.350
C00574=1014.146,215.802,-139.607,-24.382,21.399,-41.348
C00575=1014.148,216.045,-139.634,-24.383,21.398,-41.346
C00576=1014.150,216.288,-139.661,-24.383,21.398,-41.346
C00577=1014.152,216.531,-139.688,-24.383,21.398,-41.344
C00578=1014.154,216.772,-139.715,-24.383,21.398,-41.342
C00579=1014.156,217.022,-139.743,-24.383,21.399,-41.341
C00580=1014.158,217.270,-139.771,-24.384,21.398,-41.339
C00581=1014.160,217.518,-139.799,-24.384,21.397,-41.339
C00582=1014.162,217.767,-139.826,-24.384,21.397,-41.337
C00583=1014.165,218.015,-139.854,-24.384,21.398,-41.335
C00584=1014.166,218.264,-139.882,-24.384,21.398,-41.333
C00585=1014.168,218.512,-139.910,-24.385,21.397,-41.332
C00586=1014.170,218.760,-139.938,-24.385,21.397,-41.330
C00587=1014.173,219.009,-139.965,-24.385,21.397,-41.330
C00588=1014.174,219.257,-139.993,-24.385,21.397,-41.328
C00589=1014.177,219.505,-140.021,-24.385,21.397,-41.326
C00590=1014.178,219.754,-140.049,-24.386,21.397,-41.324
C00591=1014.181,220.003,-140.077,-24.386,21.397,-41.323
C00592=1014.182,220.251,-140.105,-24.386,21.397,-41.321
C00593=1014.185,220.499,-140.132,-24.386,21.396,-41.320
C00594=1014.187,220.748,-140.160,-24.386,21.396,-41.318
C00595=1014.189,220.996,-140.188,-24.387,21.397,-41.317
C00596=1014.191,221.244,-140.216,-24.387,21.396,-41.315
C00597=1014.193,221.494,-140.244,-24.387,21.396,-41.313
C00598=1014.196,221.742,-140.272,-24.388,21.396,-41.311
C00599=1014.197,221.984,-140.300,-24.388,21.397,-41.310
C00600=1014.200,222.227,-140.327,-24.388,21.396,-41.309
C00601=1014.202,222.469,-140.354,-24.388,21.395,-41.308
C00602=1014.204,222.713,-140.382,-24.388,21.395,-41.306
C00603=1014.206,222.956,-140.409,-24.389,21.396,-41.304
C00604=1014.209,223.199,-140.436,-24.389,21.396,-41.302
C00605=1014.210,223.442,-140.464,-24.389,21.395,-41.300
C00606=1014.213,223.684,-140.491,-24.389,21.395,-41.300
C00607=1014.215,223.932,-140.518,-24.389,21.394,-41.298
C00608=1014.217,224.181,-140.547,-24.390,21.395,-41.297
C00609=1014.220,224.429,-140.575,-24.390,21.395,-41.295
C00610=1014.222,224.678,-140.603,-24.390,21.395,-41.293
C00611=1014.224,224.926,-140.630,-24.390,21.394,-41.291
C00612=1014.226,225.175,-140.659,-24.391,21.394,-41.289
C00613=1014.228,225.423,-140.687,-24.391,21.395,-41.288
C00614=1014.231,225.672,-140.715,-24.391,21.395,-41.286
C00615=1014.233,225.920,-140.743,-24.391,21.394,-41.285
C00616=1014.235,226.168,-140.771,-24.391,21.393,-41.284
C00617=1014.238,226.416,-140.800,-24.392,21.393,-41.282
C00618=1014.240,226.664,-140.827,-24.392,21.394,-41.280
C00619=1014.242,226.913,-140.856,-24.392,21.394,-41.278
C00620=1014.245,227.161,-140.884,-24.393,21.393,-41.276
C00621=1014.247,227.410,-140.912,-24.393,21.393,-41.275
C00622=1014.249,227.658,-140.940,-24.393,21.393,-41.273
C00623=1014.251,227.907,-140.969,-24.393,21.394,-41.271
C00624=1014.254,228.155,-140.997,-24.394,21.393,-41.269
C00625=1014.256,228.404,-141.025,-24.394,21.393,-41.267
C00626=1014.259,228.652,-141.053,-24.394,21.393,-41.266
C00627=1014.261,228.895,-141.080,-24.394,21.392,-41.265
C00628=1014.263,229.138,-141.108,-24.394,21.392,-41.263
C00629=1014.266,229.381,-141.136,-24.395,21.392,-41.262
C00630=1014.267,229.624,-141.163,-24.395,21.392,-41.260
C00631=1014.270,229.867,-141.191,-24.395,21.392,-41.258
C00632=1014.273,230.109,-141.218,-24.395,21.392,-41.256
C00633=1014.274,230.352,-141.246,-24.396,21.392,-41.254
C00634=1014.278,230.595,-141.274,-24.396,21.391,-41.252
C00635=1014.280,230.844,-141.303,-24.396,21.392,-41.251
C00636=1014.282,231.092,-141.331,-24.396,21.392,-41.249
C00637=1014.284,231.341,-141.359,-24.397,21.392,-41.247
C00638=1014.287,231.588,-141.387,-24.397,21.391,-41.245
C00639=1014.289,231.837,-141.416,-24.397,21.391,-41.243
C00640=1014.292,232.086,-141.444,-24.397,21.391,-41.242
C00641=1014.295,232.333,-141.472,-24.398,21.391,-41.240
C00642=1014.297,232.582,-141.501,-24.398,21.390,-41.238
C00643=1014.300,232.831,-141.529,-24.398,21.391,-41.236
C00644=1014.301,233.079,-141.557,-24.399,21.391,-41.234
C00645=1014.305,233.327,-141.586,-24.399,21.391,-41.233
C00646=1014.307,233.576,-141.615,-24.399,21.390,-41.231
C00647=1014.309,233.824,-141.642,-24.399,21.390,-41.229
C00648=1014.312,234.073,-141.671,-24.400,21.390,-41.227
C00649=1014.315,234.321,-141.700,-24.400,21.390,-41.225
C00650=1014.317,234.569,-141.728,-24.400,21.390,-41.223
C00651=1014.319,234.817,-141.756,-24.400,21.389,-41.221
C00652=1014.322,235.066,-141.785,-24.401,21.389,-41.219
C00653=1014.325,235.314,-141.813,-24.401,21.389,-41.218
C00654=1014.327,235.563,-141.842,-24.401,21.390,-41.216
C00655=1014.330,235.805,-141.870,-24.401,21.389,-41.214
C00656=1014.333,236.048,-141.898,-24.402,21.389,-41.212
C00657=1014.335,236.292,-141.926,-24.402,21.389,-41.210
C00658=1014.337,236.534,-141.953,-24.402,21.389,-41.209
C00659=1014.340,236.777,-141.982,-24.402,21.388,-41.207
C00660=1014.343,237.020,-142.009,-24.403,21.388,-41.205
C00661=1014.345,237.264,-142.037,-24.403,21.388,-41.203
C00662=1014.348,237.506,-142.065,-24.403,21.388,-41.201
C00663=1014.350,237.755,-142.094,-24.403,21.388,-41.199
C00664=1014.353,238.003,-142.122,-24.404,21.387,-41.197
C00665=1014.355,238.252,-142.151,-24.404,21.387,-41.195
C00666=1014.358,238.500,-142.180,-24.405,21.388,-41.192
C00667=1014.361,238.749,-142.209,-24.405,21.387,-41.190
C00668=1014.363,238.996,-142.237,-24.405,21.387,-41.188
C00669=1014.366,239.245,-142.266,-24.405,21.387,-41.186
C00670=1014.369,239.493,-142.294,-24.406,21.387,-41.184
C00671=1014.371,239.742,-142.323,-24.406,21.386,-41.183
C00672=1014.374,239.990,-142.352,-24.406,21.386,-41.181
C00673=1014.377,240.238,-142.381,-24.406,21.386,-41.179
C00674=1014.380,240.486,-142.410,-24.407,21.386,-41.177
C00675=1014.382,240.735,-142.438,-24.407,21.386,-41.174
C00676=1014.385,240.983,-142.467,-24.407,21.386,-41.172
C00677=1014.388,241.232,-142.496,-24.408,21.386,-41.170
C00678=1014.391,241.480,-142.525,-24.408,21.386,-41.168
C00679=1014.393,241.728,-142.554,-24.408,21.385,-41.166
C00680=1014.396,241.976,-142.582,-24.408,21.385,-41.164
C00681=1014.398,242.225,-142.611,-24.409,21.385,-41.162
C00682=1014.401,242.473,-142.639,-24.409,21.385,-41.159
C00683=1014.404,242.716,-142.668,-24.410,21.385,-41.157
C00684=1014.407,242.959,-142.695,-24.410,21.385,-41.155
C00685=1014.409,243.202,-142.724,-24.410,21.385,-41.153
C00686=1014.413,243.446,-142.752,-24.410,21.384,-41.151
C00687=1014.415,243.689,-142.781,-24.411,21.384,-41.150
C00688=1014.419,243.932,-142.809,-24.411,21.384,-41.148
C00689=1014.421,244.175,-142.838,-24.411,21.384,-41.144
C00690=1014.424,244.418,-142.866,-24.412,21.384,-41.143
C00691=1014.426,244.667,-142.895,-24.412,21.384,-41.141
C00692=1014.430,244.915,-142.923,-24.412,21.384,-41.139
C00693=1014.432,245.163,-142.953,-24.412,21.384,-41.137
C00694=1014.435,245.411,-142.981,-24.413,21.384,-41.134
C00695=1014.438,245.659,-143.011,-24.413,21.384,-41.132
C00696=1014.441,245.908,-143.039,-24.413,21.383,-41.129
C00697=1014.444,246.156,-143.068,-24.414,21.382,-41.127
C00698=1014.447,246.404,-143.097,-24.414,21.382,-41.126
C00699=1014.449,246.652,-143.126,-24.414,21.383,-41.122
C00700=1014.452,246.901,-143.156,-24.415,21.382,-41.120
C00701=1014.456,247.149,-143.185,-24.415,21.382,-41.118
C00702=1014.458,247.398,-143.214,-24.415,21.382,-41.117
C00703=1014.461,247.646,-143.242,-24.416,21.382,-41.113
C00704=1014.464,247.895,-143.272,-24.416,21.382,-41.111
C00705=1014.467,248.143,-143.301,-24.416,21.381,-41.109
C00706=1014.469,248.391,-143.330,-24.417,21.381,-41.107
C00707=1014.473,248.639,-143.359,-24.417,21.381,-41.104
C00708=1014.476,248.888,-143.388,-24.417,21.381,-41.102
C00709=1014.479,249.136,-143.417,-24.418,21.381,-41.100
C00710=1014.482,249.384,-143.447,-24.418,21.381,-41.098
C00711=1014.486,249.627,-143.475,-24.418,21.381,-41.095
C00712=1014.488,249.871,-143.503,-24.419,21.381,-41.093
C00713=1014.490,250.114,-143.532,-24.419,21.380,-41.091
C00714=1014.494,250.357,-143.561,-24.419,21.380,-41.089
C00715=1014.497,250.600,-143.590,-24.420,21.380,-41.085
C00716=1014.499,250.843,-143.619,-24.420,21.380,-41.084
C00717=1014.503,251.087,-143.647,-24.420,21.380,-41.082
C00718=1014.507,251.450,-143.689,-24.421,21.379,-41.078
C00719=1014.510,251.699,-143.719,-24.421,21.379,-41.076
C00720=1014.514,251.947,-143.748,-24.422,21.379,-41.073
C00721=1014.516,252.196,-143.777,-24.422,21.379,-41.071
C00722=1014.519,252.444,-143.807,-24.422,21.378,-41.068
C00723=1014.523,252.692,-143.837,-24.423,21.378,-41.065
C00724=1014.525,252.940,-143.866,-24.423,21.378,-41.063
C00725=1014.529,253.188,-143.895,-24.423,21.378,-41.061
C00726=1014.532,253.437,-143.924,-24.424,21.378,-41.058
C00727=1014.535,253.685,-143.953,-24.424,21.377,-41.056
C00728=1014.538,253.933,-143.983,-24.424,21.377,-41.054
C00729=1014.542,254.181,-144.012,-24.425,21.378,-41.051
C00730=1014.544,254.430,-144.042,-24.425,21.377,-41.049
C00731=1014.547,254.679,-144.072,-24.426,21.378,-41.045
C00732=1014.551,254.926,-144.101,-24.426,21.377,-41.043
C00733=1014.553,255.174,-144.130,-24.426,21.376,-41.041
C00734=1014.557,255.423,-144.160,-24.427,21.377,-41.038
C00735=1014.560,255.671,-144.189,-24.427,21.377,-41.036
C00736=1014.563,255.919,-144.219,-24.427,21.376,-41.034
C00737=1014.567,256.168,-144.248,-24.428,21.376,-41.030
C00738=1014.570,256.415,-144.278,-24.428,21.376,-41.028
C00739=1014.573,256.644,-144.306,-24.428,21.376,-41.025
C00740=1014.576,256.872,-144.333,-24.429,21.376,-41.023
C00741=1014.578,257.100,-144.360,-24.429,21.376,-41.021
C00742=1014.581,257.329,-144.387,-24.429,21.375,-41.019
C00743=1014.584,257.557,-144.414,-24.430,21.375,-41.016
C00744=1014.588,257.786,-144.441,-24.430,21.375,-41.014
C00745=1014.590,258.014,-144.468,-24.430,21.375,-41.012
C00746=1014.605,259.234,-144.618,-24.552,21.323,-40.170
C00747=1014.607,259.513,-144.655,-24.587,21.310,-39.930
C00748=1014.609,259.794,-144.692,-24.622,21.298,-39.688
C00749=1014.610,260.073,-144.729,-24.658,21.287,-39.446
C00750=1014.610,260.353,-144.766,-24.693,21.275,-39.204
C00751=1014.611,260.601,-144.802,-24.726,21.267,-38.987
C00752=1014.612,260.848,-144.836,-24.758,21.259,-38.770
C00753=1014.611,261.096,-144.871,-24.790,21.252,-38.553
C00754=1014.610,261.343,-144.907,-24.823,21.244,-38.335
C00755=1014.608,261.622,-144.948,-24.860,21.238,-38.088
C00756=1014.607,261.901,-144.990,-24.897,21.232,-37.841
C00757=1014.604,262.181,-145.032,-24.935,21.227,-37.593
C00758=1014.603,262.459,-145.076,-24.973,21.223,-37.345
C00759=1014.600,262.707,-145.115,-25.006,21.220,-37.124
C00760=1014.597,262.954,-145.154,-25.040,21.217,-36.903
C00761=1014.593,263.200,-145.193,-25.074,21.216,-36.681
C00762=1014.590,263.447,-145.233,-25.108,21.215,-36.458
C00763=1014.585,263.726,-145.280,-25.147,21.216,-36.205
C00764=1014.580,264.006,-145.326,-25.186,21.217,-35.952
C00765=1014.574,264.284,-145.374,-25.226,21.219,-35.699
C00766=1014.568,264.563,-145.422,-25.265,21.221,-35.444
C00767=1014.563,264.809,-145.465,-25.300,21.225,-35.219
C00768=1014.557,265.056,-145.508,-25.335,21.229,-34.991
C00769=1014.550,265.302,-145.552,-25.370,21.233,-34.766
C00770=1014.543,265.548,-145.597,-25.406,21.239,-34.538
C00771=1014.535,265.826,-145.648,-25.446,21.246,-34.279
C00772=1014.526,266.105,-145.700,-25.487,21.254,-34.021
C00773=1014.518,266.384,-145.753,-25.527,21.264,-33.760
C00774=1014.508,266.662,-145.806,-25.568,21.275,-33.499
C00775=1014.499,266.908,-145.853,-25.604,21.284,-33.268
C00776=1014.490,267.153,-145.901,-25.641,21.295,-33.037
C00777=1014.481,267.398,-145.950,-25.677,21.306,-32.805
C00778=1014.471,267.644,-145.999,-25.714,21.319,-32.571
C00779=1014.459,267.922,-146.054,-25.755,21.334,-32.305
C00780=1014.447,268.200,-146.112,-25.797,21.350,-32.039
C00781=1014.436,268.479,-146.170,-25.839,21.367,-31.772
C00782=1014.422,268.757,-146.228,-25.881,21.386,-31.502
C00783=1014.410,269.002,-146.279,-25.918,21.402,-31.266
C00784=1014.398,269.246,-146.331,-25.955,21.420,-31.029
C00785=1014.385,269.490,-146.385,-25.992,21.439,-30.789
C00786=1014.371,269.734,-146.437,-26.030,21.459,-30.551
C00787=1014.357,270.013,-146.499,-26.072,21.483,-30.277
C00788=1014.342,270.291,-146.562,-26.115,21.507,-30.003
C00789=1014.325,270.569,-146.624,-26.158,21.533,-29.728
C00790=1014.308,270.847,-146.688,-26.201,21.560,-29.450
C00791=1014.294,271.090,-146.744,-26.238,21.585,-29.208
C00792=1014.279,271.333,-146.800,-26.276,21.610,-28.964
C00793=1014.263,271.576,-146.858,-26.314,21.637,-28.720
C00794=1014.246,271.819,-146.916,-26.351,21.664,-28.476
C00795=1014.229,272.097,-146.983,-26.395,21.697,-28.194
C00796=1014.209,272.375,-147.050,-26.438,21.731,-27.910
C00797=1014.189,272.653,-147.117,-26.481,21.766,-27.626
C00798=1014.168,272.931,-147.187,-26.525,21.803,-27.342
C00799=1014.150,273.173,-147.247,-26.562,21.835,-27.092
C00800=1014.132,273.414,-147.308,-26.600,21.869,-26.841
C00801=1014.113,273.656,-147.370,-26.638,21.904,-26.589
C00802=1014.094,273.898,-147.432,-26.676,21.940,-26.336
C00803=1014.071,274.176,-147.504,-26.720,21.983,-26.043
C00804=1014.048,274.453,-147.577,-26.763,22.027,-25.750
C00805=1014.026,274.730,-147.651,-26.807,22.073,-25.453
C00806=1014.001,275.008,-147.726,-26.851,22.119,-25.156
C00807=1013.980,275.248,-147.790,-26.889,22.162,-24.896
C00808=1013.959,275.489,-147.856,-26.927,22.204,-24.635
C00809=1013.936,275.729,-147.923,-26.965,22.250,-24.373
C00810=1013.913,275.969,-147.989,-27.003,22.295,-24.109
C00811=1013.888,276.247,-148.066,-27.046,22.349,-23.804
C00812=1013.860,276.523,-148.145,-27.090,22.404,-23.496
C00813=1013.833,276.800,-148.224,-27.134,22.462,-23.186
C00814=1013.806,277.078,-148.303,-27.177,22.521,-22.877
C00815=1013.781,277.316,-148.374,-27.215,22.572,-22.606
C00816=1013.756,277.555,-148.444,-27.252,22.626,-22.334
C00817=1013.731,277.794,-148.515,-27.290,22.681,-22.062
C00818=1013.705,278.033,-148.586,-27.327,22.738,-21.787
C00819=1013.675,278.309,-148.669,-27.370,22.804,-21.468
C00820=1013.645,278.586,-148.754,-27.413,22.873,-21.147
C00821=1013.613,278.862,-148.839,-27.456,22.942,-20.824
C00822=1013.581,279.138,-148.924,-27.498,23.014,-20.499
C00823=1013.553,279.376,-148.998,-27.534,23.077,-20.218
C00824=1013.525,279.612,-149.073,-27.570,23.142,-19.936
C00825=1013.496,279.849,-149.148,-27.606,23.208,-19.653
C00826=1013.467,280.087,-149.224,-27.642,23.276,-19.366
C00827=1013.432,280.363,-149.313,-27.684,23.356,-19.030
C00828=1013.398,280.638,-149.403,-27.725,23.440,-18.691
C00829=1013.363,280.914,-149.494,-27.766,23.526,-18.349
C00830=1013.326,281.189,-149.586,-27.807,23.613,-18.004
C00831=1013.295,281.425,-149.665,-27.842,23.690,-17.706
C00832=1013.262,281.660,-149.744,-27.877,23.768,-17.406
C00833=1013.231,281.895,-149.824,-27.911,23.848,-17.104
C00834=1013.199,282.129,-149.905,-27.945,23.930,-16.800
C00835=1013.161,282.404,-150.000,-27.985,24.028,-16.440
C00836=1013.121,282.679,-150.096,-28.024,24.129,-16.077
C00837=1013.081,282.954,-150.193,-28.062,24.232,-15.713
C00838=1013.040,283.228,-150.291,-28.100,24.338,-15.343
C00839=1013.006,283.461,-150.375,-28.132,24.429,-15.026
C00840=1012.970,283.694,-150.459,-28.164,24.524,-14.708
C00841=1012.935,283.927,-150.544,-28.195,24.619,-14.388
C00842=1012.899,284.160,-150.629,-28.226,24.716,-14.065
C00843=1012.856,284.434,-150.731,-28.261,24.835,-13.680
C00844=1012.813,284.707,-150.833,-28.296,24.955,-13.292
C00845=1012.768,284.981,-150.937,-28.330,25.079,-12.901
C00846=1012.723,285.255,-151.040,-28.364,25.204,-12.507
C00847=1012.684,285.485,-151.129,-28.391,25.314,-12.171
C00848=1012.645,285.716,-151.218,-28.418,25.425,-11.832
C00849=1012.606,285.946,-151.308,-28.444,25.537,-11.492
C00850=1012.567,286.175,-151.399,-28.470,25.652,-11.148
C00851=1012.518,286.448,-151.507,-28.499,25.792,-10.737
C00852=1012.470,286.721,-151.616,-28.527,25.936,-10.320
C00853=1012.421,286.993,-151.726,-28.555,26.082,-9.899
C00854=1012.371,287.265,-151.837,-28.581,26.233,-9.471
C00855=1012.329,287.493,-151.932,-28.602,26.363,-9.109
C00856=1012.286,287.720,-152.026,-28.622,26.494,-8.743
C00857=1012.243,287.948,-152.121,-28.641,26.630,-8.372
C00858=1012.200,288.175,-152.217,-28.659,26.768,-7.997
C00859=1012.147,288.446,-152.332,-28.679,26.937,-7.545
C00860=1012.093,288.717,-152.447,-28.698,27.110,-7.087
C00861=1012.039,288.987,-152.565,-28.715,27.285,-6.624
C00862=1011.985,289.258,-152.683,-28.730,27.467,-6.153
C00863=1011.938,289.482,-152.783,-28.742,27.622,-5.757
C00864=1011.892,289.707,-152.882,-28.752,27.779,-5.357
C00865=1011.844,289.931,-152.983,-28.760,27.939,-4.952
C00866=1011.797,290.155,-153.084,-28.767,28.103,-4.544
C00867=1011.739,290.424,-153.207,-28.773,28.305,-4.046
C00868=1011.679,290.693,-153.330,-28.777,28.512,-3.541
C00869=1011.620,290.961,-153.455,-28.778,28.722,-3.030
C00870=1011.560,291.229,-153.580,-28.777,28.937,-2.514
C00871=1011.510,291.451,-153.686,-28.773,29.120,-2.080
C00872=1011.459,291.672,-153.791,-28.768,29.306,-1.642
C00873=1011.408,291.892,-153.898,-28.760,29.495,-1.198
C00874=1011.355,292.112,-154.004,-28.751,29.688,-0.751
C00875=1011.291,292.380,-154.135,-28.736,29.926,-0.203
C00876=1011.227,292.646,-154.266,-28.717,30.168,0.353
C00877=1011.163,292.911,-154.399,-28.695,30.417,0.916
C00878=1011.096,293.177,-154.532,-28.669,30.673,1.490
C00879=1011.042,293.394,-154.644,-28.645,30.886,1.967
C00880=1010.986,293.611,-154.755,-28.617,31.104,2.450
C00881=1010.931,293.828,-154.867,-28.586,31.327,2.940
C00882=1010.874,294.044,-154.979,-28.552,31.552,3.436
C00883=1010.805,294.307,-155.118,-28.506,31.835,4.050
C00884=1010.734,294.571,-155.258,-28.455,32.122,4.672
C00885=1010.664,294.833,-155.399,-28.398,32.416,5.305
C00886=1010.591,295.095,-155.542,-28.335,32.716,5.947
C00887=1010.532,295.308,-155.658,-28.280,32.966,6.479
C00888=1010.472,295.522,-155.776,-28.220,33.220,7.016
C00889=1010.411,295.734,-155.894,-28.156,33.478,7.560
C00890=1010.350,295.945,-156.013,-28.087,33.739,8.111
C00891=1010.274,296.206,-156.160,-27.996,34.069,8.801
C00892=1010.198,296.465,-156.310,-27.897,34.404,9.500
C00893=1010.120,296.724,-156.460,-27.790,34.746,10.213
C00894=1010.042,296.982,-156.611,-27.675,35.094,10.935
C00895=1009.978,297.191,-156.733,-27.576,35.380,11.529
C00896=1009.913,297.398,-156.858,-27.470,35.670,12.129
C00897=1009.848,297.605,-156.983,-27.359,35.965,12.738
C00898=1009.782,297.812,-157.107,-27.241,36.263,13.354
C00899=1009.699,298.068,-157.265,-27.085,36.641,14.134
C00900=1009.616,298.323,-157.423,-26.918,37.024,14.926
C00901=1009.531,298.578,-157.582,-26.741,37.414,15.733
C00902=1009.446,298.832,-157.743,-26.551,37.810,16.553
C00903=1009.377,299.034,-157.873,-26.391,38.132,17.220
C00904=1009.307,299.237,-158.002,-26.221,38.458,17.898
C00905=1009.237,299.439,-158.134,-26.044,38.788,18.586
C00906=1009.166,299.639,-158.265,-25.857,39.121,19.283
///RCONF 0,0,0,0,0,0,0,0,0,0,0,0,0,0,0,0,0,0,0,0,0,0,0,0
C00907=1009.077,299.890,-158.432,-25.611,39.544,20.170
C00908=1008.986,300.141,-158.600,-25.349,39.974,21.077
C00909=1008.894,300.391,-158.770,-25.071,40.409,21.999
C00910=1008.801,300.640,-158.940,-24.778,40.847,22.938
C00911=1008.727,300.836,-159.076,-24.533,41.199,23.695
C00912=1008.652,301.032,-159.212,-24.278,41.553,24.463
C00913=1008.578,301.227,-159.350,-24.010,41.911,25.245
C00914=1008.502,301.422,-159.489,-23.731,42.271,26.037
C00915=1008.404,301.668,-159.666,-23.359,42.732,27.060
C00916=1008.306,301.912,-159.844,-22.967,43.196,28.105
C00917=1008.207,302.157,-160.023,-22.552,43.665,29.173
C00918=1008.107,302.400,-160.203,-22.115,44.137,30.264
C00919=1008.027,302.589,-160.347,-21.757,44.508,31.133
C00920=1007.948,302.777,-160.490,-21.384,44.880,32.017
C00921=1007.867,302.966,-160.634,-20.996,45.254,32.916
C00922=1007.786,303.154,-160.779,-20.592,45.628,33.828
C00923=1007.681,303.393,-160.966,-20.052,46.107,35.019
C00924=1007.574,303.632,-161.154,-19.485,46.587,36.235
C00925=1007.468,303.870,-161.344,-18.890,47.066,37.479
C00926=1007.360,304.105,-161.536,-18.265,47.545,38.750
C00927=1007.276,304.287,-161.684,-17.761,47.914,39.754
C00928=1007.190,304.469,-161.834,-17.237,48.283,40.777
C00929=1007.105,304.650,-161.985,-16.695,48.650,41.816
C00930=1007.019,304.830,-162.136,-16.132,49.015,42.875
C00931=1006.906,305.062,-162.334,-15.372,49.485,44.275
C00932=1006.793,305.294,-162.533,-14.578,49.950,45.708
C00933=1006.678,305.524,-162.732,-13.751,50.408,47.169
C00934=1006.562,305.752,-162.934,-12.888,50.859,48.662
C00935=1006.473,305.926,-163.090,-12.202,51.199,49.829
C00936=1006.383,306.099,-163.245,-11.496,51.534,51.012
C00937=1006.292,306.273,-163.403,-10.769,51.863,52.214
C00938=1006.200,306.445,-163.560,-10.019,52.186,53.436
C00939=1006.080,306.669,-163.768,-9.002,52.599,55.068
C00940=1005.958,306.892,-163.977,-7.948,53.000,56.733
C00941=1005.836,307.113,-164.187,-6.854,53.388,58.434
C00942=1005.712,307.333,-164.398,-5.724,53.761,60.165
C00943=1005.619,307.499,-164.560,-4.837,54.035,61.506
C00944=1005.523,307.665,-164.721,-3.930,54.299,62.863
C00945=1005.428,307.829,-164.885,-2.997,54.554,64.245
C00946=1005.332,307.993,-165.048,-2.047,54.798,65.640
C00947=1005.204,308.208,-165.265,-0.758,55.103,67.512
C00948=1005.075,308.421,-165.484,0.567,55.388,69.414
C00949=1004.944,308.633,-165.704,1.921,55.651,71.337
C00950=1004.788,308.884,-165.967,3.574,55.935,73.662
C00951=1004.763,308.924,-166.010,3.845,55.978,74.040
C00952=1005.166,309.094,-166.457,4.755,56.114,75.307
C00953=1005.301,308.879,-166.229,3.305,55.891,73.285
C00954=1005.431,308.669,-166.008,1.921,55.651,71.337
C00955=1005.561,308.457,-165.788,0.567,55.388,69.414
C00956=1005.691,308.242,-165.570,-0.758,55.103,67.512
C00957=1005.819,308.028,-165.352,-2.047,54.798,65.640
C00958=1005.915,307.864,-165.189,-2.997,54.554,64.245
C00959=1006.010,307.700,-165.025,-3.930,54.299,62.863
C00960=1006.106,307.535,-164.864,-4.837,54.035,61.506
C00961=1006.199,307.369,-164.702,-5.724,53.761,60.165
C00962=1006.323,307.148,-164.490,-6.854,53.388,58.434
C00963=1006.445,306.927,-164.280,-7.948,53.000,56.733
C00964=1006.567,306.704,-164.071,-9.002,52.599,55.068
C00965=1006.687,306.480,-163.864,-10.019,52.186,53.436
C00966=1006.779,306.308,-163.706,-10.767,51.863,52.216
C00967=1006.869,306.135,-163.548,-11.496,51.534,51.012
C00968=1006.959,305.961,-163.392,-12.202,51.199,49.829
C00969=1007.048,305.787,-163.238,-12.888,50.859,48.662
C00970=1007.165,305.559,-163.036,-13.751,50.408,47.169
C00971=1007.278,305.329,-162.836,-14.578,49.950,45.708
C00972=1007.393,305.098,-162.637,-15.372,49.485,44.275
C00973=1007.505,304.866,-162.439,-16.132,49.015,42.875
C00974=1007.592,304.686,-162.288,-16.695,48.650,41.816
C00975=1007.677,304.505,-162.137,-17.237,48.283,40.777
C00976=1007.762,304.323,-161.987,-17.761,47.914,39.754
C00977=1007.846,304.141,-161.839,-18.265,47.545,38.750
C00978=1007.954,303.904,-161.648,-18.890,47.066,37.479
C00979=1008.060,303.667,-161.457,-19.485,46.587,36.235
C00980=1008.167,303.428,-161.269,-20.052,46.107,35.019
C00981=1008.272,303.189,-161.082,-20.592,45.628,33.828
C00982=1008.353,303.001,-160.937,-20.996,45.254,32.916
C00983=1008.433,302.813,-160.793,-21.384,44.880,32.017
C00984=1008.513,302.624,-160.650,-21.757,44.508,31.133
C00985=1008.592,302.435,-160.507,-22.115,44.137,30.264
C00986=1008.692,302.192,-160.326,-22.552,43.665,29.173
C00987=1008.791,301.947,-160.146,-22.967,43.196,28.105
C00988=1008.890,301.703,-159.968,-23.359,42.732,27.060
C00989=1008.986,301.457,-159.791,-23.731,42.271,26.037
C00990=1009.062,301.262,-159.653,-24.010,41.911,25.245
C00991=1009.137,301.067,-159.515,-24.278,41.553,24.463
C00992=1009.212,300.871,-159.378,-24.533,41.199,23.695
C00993=1009.286,300.675,-159.243,-24.778,40.847,22.938
C00994=1009.379,300.426,-159.071,-25.071,40.409,21.999
C00995=1009.470,300.176,-158.902,-25.349,39.974,21.077
C00996=1009.561,299.926,-158.735,-25.611,39.544,20.170
///RCONF 0,0,0,0,1,0,0,0,0,0,0,0,0,0,0,0,0,0,0,0,0,0,0,0
C00997=1009.650,299.674,-158.567,-25.857,39.121,19.283
C00998=1009.721,299.473,-158.435,-26.044,38.788,18.586
C00999=1009.791,299.272,-158.304,-26.221,38.458,17.898
C01000=1009.860,299.070,-158.174,-26.391,38.132,17.220
C01001=1009.930,298.868,-158.045,-26.551,37.810,16.553
C01002=1010.015,298.613,-157.884,-26.741,37.414,15.733
C01003=1010.100,298.359,-157.724,-26.918,37.024,14.926
C01004=1010.183,298.103,-157.566,-27.085,36.641,14.134
C01005=1010.266,297.847,-157.409,-27.241,36.263,13.354
C01006=1010.331,297.641,-157.284,-27.359,35.965,12.738
C01007=1010.397,297.433,-157.159,-27.470,35.670,12.129
C01008=1010.461,297.225,-157.035,-27.576,35.380,11.529
C01009=1010.525,297.017,-156.912,-27.675,35.094,10.935
C01010=1010.604,296.759,-156.761,-27.790,34.746,10.213
C01011=1010.681,296.500,-156.611,-27.897,34.404,9.500
C01012=1010.758,296.241,-156.462,-27.996,34.069,8.801
C01013=1010.834,295.980,-156.315,-28.087,33.739,8.111
C01014=1010.894,295.769,-156.195,-28.156,33.478,7.560
C01015=1010.954,295.556,-156.076,-28.220,33.220,7.016
C01016=1011.014,295.344,-155.959,-28.280,32.966,6.479
C01017=1011.074,295.130,-155.843,-28.335,32.716,5.947
C01018=1011.146,294.868,-155.700,-28.398,32.417,5.306
C01019=1011.217,294.606,-155.559,-28.455,32.122,4.672
C01020=1011.287,294.343,-155.420,-28.506,31.835,4.050
C01021=1011.357,294.078,-155.279,-28.552,31.552,3.436
C01022=1011.413,293.862,-155.167,-28.586,31.327,2.940
C01023=1011.469,293.646,-155.055,-28.617,31.104,2.450
C01024=1011.524,293.429,-154.944,-28.645,30.886,1.967
C01025=1011.578,293.211,-154.833,-28.669,30.673,1.490
C01026=1011.644,292.946,-154.700,-28.695,30.417,0.916
C01027=1011.709,292.680,-154.567,-28.717,30.168,0.353
C01028=1011.774,292.414,-154.436,-28.736,29.926,-0.203
C01029=1011.837,292.147,-154.304,-28.751,29.688,-0.751
C01030=1011.889,291.927,-154.198,-28.760,29.495,-1.198
C01031=1011.940,291.707,-154.091,-28.768,29.306,-1.642
C01032=1011.992,291.485,-153.985,-28.773,29.120,-2.080
C01033=1012.041,291.264,-153.880,-28.777,28.937,-2.514
C01034=1012.102,290.996,-153.755,-28.778,28.722,-3.030
C01035=1012.162,290.728,-153.630,-28.777,28.512,-3.541
C01036=1012.220,290.459,-153.507,-28.773,28.305,-4.046
C01037=1012.278,290.190,-153.384,-28.767,28.103,-4.544
C01038=1012.325,289.966,-153.283,-28.760,27.939,-4.952
C01039=1012.373,289.741,-153.182,-28.752,27.779,-5.357
C01040=1012.419,289.517,-153.082,-28.742,27.622,-5.757
C01041=1012.466,289.292,-152.983,-28.730,27.467,-6.153
C01042=1012.520,289.022,-152.865,-28.715,27.285,-6.624
C01043=1012.574,288.752,-152.748,-28.698,27.109,-7.088
C01044=1012.627,288.481,-152.631,-28.679,26.937,-7.545
C01045=1012.680,288.210,-152.516,-28.659,26.767,-7.999
C01046=1012.724,287.982,-152.421,-28.641,26.630,-8.372
C01047=1012.767,287.755,-152.326,-28.622,26.495,-8.743
C01048=1012.810,287.527,-152.231,-28.602,26.363,-9.109
C01049=1012.851,287.299,-152.137,-28.581,26.233,-9.471
C01050=1012.902,287.028,-152.026,-28.555,26.082,-9.899
C01051=1012.950,286.755,-151.916,-28.527,25.936,-10.320
C01052=1012.999,286.483,-151.806,-28.499,25.792,-10.737
C01053=1013.047,286.210,-151.699,-28.470,25.652,-11.148
C01054=1013.086,285.981,-151.608,-28.444,25.537,-11.492
C01055=1013.126,285.750,-151.518,-28.418,25.425,-11.832
C01056=1013.164,285.520,-151.429,-28.391,25.314,-12.171
C01057=1013.202,285.289,-151.340,-28.364,25.204,-12.507
C01058=1013.247,285.015,-151.235,-28.330,25.079,-12.901
C01059=1013.292,284.743,-151.133,-28.296,24.955,-13.292
C01060=1013.335,284.468,-151.030,-28.261,24.835,-13.680
C01061=1013.379,284.195,-150.928,-28.226,24.716,-14.065
C01062=1013.414,283.962,-150.842,-28.195,24.619,-14.388
C01063=1013.450,283.729,-150.757,-28.164,24.524,-14.708
C01064=1013.485,283.496,-150.673,-28.132,24.429,-15.026
C01065=1013.520,283.263,-150.589,-28.100,24.338,-15.343
C01066=1013.560,282.988,-150.491,-28.062,24.232,-15.713
C01067=1013.600,282.714,-150.395,-28.024,24.129,-16.077
C01068=1013.639,282.439,-150.299,-27.985,24.028,-16.440
C01069=1013.677,282.164,-150.203,-27.945,23.930,-16.800
C01070=1013.710,281.930,-150.122,-27.911,23.848,-17.104
C01071=1013.742,281.694,-150.042,-27.877,23.768,-17.406
C01072=1013.774,281.459,-149.963,-27.842,23.690,-17.706
C01073=1013.804,281.224,-149.883,-27.807,23.613,-18.004
C01074=1013.841,280.949,-149.792,-27.766,23.526,-18.349
C01075=1013.876,280.673,-149.702,-27.725,23.440,-18.691
C01076=1013.911,280.397,-149.611,-27.684,23.356,-19.030
C01077=1013.945,280.122,-149.522,-27.642,23.276,-19.366
C01078=1013.975,279.885,-149.446,-27.606,23.208,-19.653
C01079=1014.004,279.647,-149.371,-27.570,23.142,-19.936
C01080=1014.031,279.410,-149.296,-27.534,23.078,-20.218
C01081=1014.058,279.173,-149.222,-27.498,23.014,-20.499
C01082=1014.091,278.897,-149.136,-27.456,22.942,-20.824
C01083=1014.122,278.621,-149.051,-27.413,22.872,-21.148
C01084=1014.152,278.344,-148.967,-27.370,22.804,-21.469
C01085=1014.183,278.066,-148.883,-27.327,22.737,-21.789
C01086=1014.208,277.828,-148.812,-27.290,22.681,-22.062
C01087=1014.234,277.590,-148.742,-27.252,22.627,-22.335
C01088=1014.259,277.351,-148.671,-27.215,22.573,-22.606
C01089=1014.282,277.112,-148.601,-27.177,22.521,-22.877
C01090=1014.311,276.835,-148.522,-27.134,22.462,-23.186
C01091=1014.338,276.558,-148.442,-27.090,22.404,-23.496
C01092=1014.365,276.281,-148.364,-27.046,22.349,-23.804
C01093=1014.391,276.004,-148.286,-27.003,22.295,-24.109
C01094=1014.413,275.764,-148.219,-26.965,22.250,-24.373
C01095=1014.436,275.523,-148.153,-26.927,22.204,-24.635
C01096=1014.456,275.283,-148.088,-26.889,22.162,-24.896
C01097=1014.478,275.042,-148.022,-26.851,22.119,-25.156
C01098=1014.502,274.765,-147.948,-26.807,22.073,-25.453
C01099=1014.525,274.487,-147.874,-26.763,22.027,-25.750
C01100=1014.548,274.209,-147.801,-26.720,21.983,-26.043
C01101=1014.570,273.933,-147.729,-26.676,21.940,-26.336
C01102=1014.590,273.691,-147.667,-26.638,21.904,-26.589
C01103=1014.608,273.449,-147.606,-26.600,21.869,-26.841
C01104=1014.626,273.207,-147.544,-26.562,21.835,-27.092
C01105=1014.644,272.966,-147.484,-26.525,21.803,-27.342
C01106=1014.665,272.688,-147.414,-26.481,21.766,-27.626
C01107=1014.685,272.410,-147.346,-26.438,21.731,-27.910
C01108=1014.704,272.132,-147.279,-26.395,21.697,-28.194
C01109=1014.722,271.853,-147.211,-26.351,21.664,-28.476
C01110=1014.738,271.611,-147.154,-26.314,21.637,-28.720
C01111=1014.755,271.368,-147.097,-26.276,21.610,-28.964
C01112=1014.770,271.125,-147.040,-26.238,21.585,-29.208
C01113=1014.784,270.881,-146.984,-26.201,21.560,-29.450
C01114=1014.800,270.604,-146.921,-26.158,21.533,-29.728
C01115=1014.817,270.325,-146.857,-26.115,21.507,-30.003
C01116=1014.832,270.047,-146.795,-26.072,21.483,-30.277
C01117=1014.846,269.769,-146.733,-26.030,21.459,-30.551
C01118=1014.860,269.524,-146.680,-25.992,21.439,-30.789
C01119=1014.872,269.280,-146.627,-25.955,21.420,-31.029
C01120=1014.884,269.036,-146.574,-25.918,21.402,-31.266
C01121=1014.896,268.792,-146.523,-25.881,21.386,-31.502
C01122=1014.909,268.513,-146.464,-25.839,21.367,-31.772
C01123=1014.921,268.235,-146.407,-25.797,21.350,-32.039
C01124=1014.933,267.957,-146.350,-25.755,21.334,-32.305
C01125=1014.945,267.678,-146.293,-25.714,21.319,-32.571
C01126=1014.955,267.433,-146.245,-25.677,21.306,-32.805
C01127=1014.964,267.187,-146.196,-25.641,21.295,-33.037
C01128=1014.972,266.942,-146.148,-25.604,21.284,-33.268
C01129=1014.981,266.697,-146.101,-25.568,21.275,-33.499
C01130=1014.991,266.418,-146.048,-25.527,21.264,-33.760
C01131=1014.999,266.139,-145.994,-25.487,21.254,-34.021
C01132=1015.008,265.860,-145.943,-25.446,21.246,-34.279
C01133=1015.016,265.581,-145.892,-25.406,21.239,-34.538
C01134=1015.022,265.336,-145.847,-25.370,21.233,-34.766
C01135=1015.029,265.089,-145.803,-25.335,21.229,-34.991
C01136=1015.035,264.844,-145.759,-25.300,21.225,-35.219
C01137=1015.041,264.597,-145.716,-25.265,21.221,-35.444
C01138=1015.046,264.318,-145.668,-25.226,21.219,-35.699
C01139=1015.052,264.040,-145.620,-25.186,21.217,-35.952
C01140=1015.057,263.760,-145.574,-25.147,21.216,-36.205
C01141=1015.062,263.481,-145.527,-25.108,21.215,-36.458
C01142=1015.065,263.235,-145.487,-25.074,21.216,-36.681
C01143=1015.068,262.987,-145.448,-25.040,21.217,-36.903
C01144=1015.072,262.740,-145.408,-25.006,21.220,-37.124
C01145=1015.074,262.494,-145.370,-24.973,21.223,-37.345
C01146=1015.076,262.215,-145.326,-24.935,21.226,-37.595
C01147=1015.078,261.935,-145.284,-24.897,21.233,-37.842
C01148=1015.079,261.656,-145.242,-24.860,21.238,-38.090
C01149=1015.080,261.376,-145.200,-24.823,21.245,-38.337
C01150=1015.082,261.129,-145.165,-24.790,21.251,-38.554
C01151=1015.082,260.882,-145.130,-24.758,21.259,-38.770
C01152=1015.082,260.634,-145.094,-24.725,21.267,-38.988
C01153=1015.080,260.386,-145.060,-24.693,21.275,-39.204
C01154=1015.080,260.107,-145.022,-24.658,21.287,-39.446
C01155=1015.079,259.827,-144.985,-24.622,21.298,-39.688
C01156=1015.077,259.548,-144.947,-24.587,21.310,-39.930
C01157=1015.074,259.268,-144.911,-24.551,21.322,-40.171
C01158=1015.060,258.032,-144.759,-24.430,21.375,-41.012
C01159=1015.057,257.789,-144.730,-24.430,21.375,-41.014
C01160=1015.053,257.545,-144.701,-24.429,21.375,-41.018
C01161=1015.050,257.302,-144.672,-24.429,21.376,-41.019
C01162=1015.047,257.059,-144.643,-24.429,21.376,-41.021
C01163=1015.044,256.815,-144.614,-24.428,21.375,-41.025
C01164=1015.040,256.572,-144.585,-24.428,21.376,-41.027
C01165=1015.037,256.328,-144.556,-24.428,21.377,-41.029
C01166=1015.034,256.081,-144.526,-24.427,21.376,-41.032
C01167=1015.030,255.832,-144.497,-24.427,21.376,-41.034
C01168=1015.027,255.584,-144.467,-24.426,21.376,-41.037
C01169=1015.024,255.336,-144.437,-24.426,21.377,-41.040
C01170=1015.021,255.087,-144.408,-24.426,21.377,-41.042
C01171=1015.017,254.840,-144.379,-24.425,21.377,-41.045
C01172=1015.014,254.591,-144.349,-24.425,21.377,-41.047
C01173=1015.011,254.343,-144.320,-24.425,21.377,-41.049
C01174=1015.008,254.094,-144.290,-24.424,21.378,-41.052
C01175=1015.004,253.847,-144.261,-24.424,21.378,-41.054
C01176=1015.002,253.598,-144.231,-24.424,21.378,-41.058
C01177=1014.998,253.350,-144.202,-24.423,21.378,-41.060
C01178=1014.995,253.101,-144.173,-24.423,21.378,-41.061
C01179=1014.991,252.853,-144.143,-24.423,21.378,-41.065
C01180=1014.989,252.605,-144.114,-24.422,21.379,-41.067
C01181=1014.986,252.357,-144.084,-24.422,21.379,-41.069
C01182=1014.982,252.108,-144.055,-24.421,21.378,-41.072
C01183=1014.980,251.860,-144.026,-24.421,21.379,-41.074
C01184=1014.977,251.612,-143.997,-24.421,21.380,-41.076
C01185=1014.974,251.364,-143.967,-24.421,21.380,-41.078
C01186=1014.970,251.107,-143.937,-24.420,21.380,-41.082
C01187=1014.967,250.850,-143.906,-24.420,21.380,-41.084
C01188=1014.964,250.594,-143.876,-24.419,21.379,-41.087
C01189=1014.960,250.337,-143.846,-24.419,21.380,-41.089
C01190=1014.958,250.089,-143.817,-24.419,21.381,-41.091
C01191=1014.955,249.841,-143.788,-24.419,21.381,-41.093
C01192=1014.951,249.592,-143.758,-24.418,21.380,-41.096
C01193=1014.948,249.344,-143.730,-24.418,21.381,-41.098
C01194=1014.946,249.096,-143.700,-24.418,21.381,-41.100
C01195=1014.942,248.849,-143.671,-24.417,21.380,-41.103
C01196=1014.940,248.600,-143.641,-24.417,21.382,-41.106
C01197=1014.936,248.352,-143.612,-24.417,21.382,-41.108
C01198=1014.933,248.103,-143.583,-24.416,21.382,-41.109
C01199=1014.930,247.855,-143.554,-24.416,21.382,-41.113
C01200=1014.927,247.607,-143.525,-24.415,21.382,-41.115
C01201=1014.924,247.359,-143.497,-24.415,21.382,-41.117
C01202=1014.921,247.119,-143.468,-24.415,21.382,-41.118
C01203=1014.918,246.880,-143.440,-24.415,21.382,-41.120
C01204=1014.915,246.641,-143.412,-24.414,21.382,-41.124
C01205=1014.913,246.402,-143.384,-24.414,21.382,-41.126
C01206=1014.910,246.163,-143.356,-24.414,21.382,-41.127
C01207=1014.907,245.923,-143.328,-24.413,21.384,-41.130
C01208=1014.904,245.684,-143.300,-24.413,21.384,-41.132
C01209=1014.902,245.445,-143.272,-24.413,21.384,-41.134
C01210=1014.898,245.197,-143.243,-24.412,21.384,-41.137
C01211=1014.896,244.949,-143.214,-24.412,21.384,-41.139
C01212=1014.893,244.700,-143.186,-24.412,21.384,-41.141
C01213=1014.890,244.452,-143.156,-24.412,21.384,-41.143
C01214=1014.887,244.209,-143.128,-24.411,21.384,-41.144
C01215=1014.885,243.966,-143.100,-24.411,21.384,-41.148
C01216=1014.881,243.722,-143.071,-24.411,21.384,-41.150
C01217=1014.879,243.479,-143.043,-24.410,21.384,-41.151
C01218=1014.876,243.236,-143.015,-24.410,21.385,-41.153
C01219=1014.873,242.993,-142.986,-24.410,21.385,-41.155
C01220=1014.870,242.750,-142.959,-24.410,21.385,-41.157
C01221=1014.868,242.507,-142.930,-24.409,21.385,-41.159
C01222=1014.865,242.259,-142.902,-24.409,21.385,-41.162
C01223=1014.862,242.010,-142.872,-24.408,21.385,-41.164
C01224=1014.859,241.762,-142.843,-24.408,21.385,-41.166
C01225=1014.857,241.513,-142.815,-24.408,21.386,-41.168
C01226=1014.853,241.265,-142.786,-24.408,21.386,-41.170
C01227=1014.851,241.017,-142.757,-24.407,21.386,-41.172
C01228=1014.848,240.769,-142.729,-24.407,21.386,-41.174
C01229=1014.845,240.520,-142.699,-24.407,21.386,-41.177
C01230=1014.842,240.272,-142.671,-24.406,21.386,-41.179
C01231=1014.840,240.023,-142.642,-24.406,21.386,-41.181
C01232=1014.837,239.775,-142.613,-24.406,21.386,-41.183
C01233=1014.834,239.527,-142.584,-24.406,21.387,-41.184
C01234=1014.831,239.279,-142.556,-24.405,21.387,-41.186
C01235=1014.829,239.030,-142.527,-24.405,21.387,-41.188
C01236=1014.826,238.782,-142.498,-24.405,21.387,-41.190
C01237=1014.823,238.534,-142.470,-24.405,21.388,-41.192
C01238=1014.821,238.286,-142.441,-24.404,21.387,-41.195
C01239=1014.818,238.037,-142.413,-24.404,21.387,-41.197
C01240=1014.815,237.789,-142.384,-24.403,21.388,-41.199
C01241=1014.812,237.540,-142.356,-24.403,21.388,-41.201
C01242=1014.810,237.297,-142.327,-24.403,21.388,-41.203
C01243=1014.807,237.054,-142.299,-24.403,21.388,-41.205
C01244=1014.805,236.811,-142.271,-24.402,21.388,-41.207
C01245=1014.802,236.568,-142.243,-24.402,21.389,-41.209
C01246=1014.800,236.325,-142.215,-24.402,21.389,-41.210
C01247=1014.797,236.082,-142.187,-24.402,21.389,-41.212
C01248=1014.794,235.839,-142.160,-24.401,21.389,-41.214
C01249=1014.792,235.596,-142.131,-24.401,21.390,-41.216
C01250=1014.789,235.348,-142.103,-24.401,21.389,-41.218
C01251=1014.787,235.099,-142.075,-24.401,21.389,-41.219
C01252=1014.783,234.851,-142.046,-24.400,21.389,-41.221
C01253=1014.782,234.603,-142.017,-24.400,21.390,-41.223
C01254=1014.778,234.355,-141.989,-24.400,21.390,-41.225
C01255=1014.776,234.106,-141.960,-24.400,21.390,-41.227
C01256=1014.773,233.857,-141.932,-24.399,21.390,-41.229
C01257=1014.772,233.609,-141.904,-24.399,21.390,-41.231
C01258=1014.768,233.361,-141.875,-24.399,21.391,-41.233
C01259=1014.765,233.112,-141.847,-24.399,21.391,-41.234
C01260=1014.764,232.864,-141.819,-24.398,21.391,-41.236
C01261=1014.761,232.616,-141.790,-24.398,21.390,-41.238
C01262=1014.758,232.367,-141.761,-24.398,21.391,-41.240
C01263=1014.755,232.119,-141.733,-24.397,21.391,-41.242
C01264=1014.754,231.870,-141.705,-24.397,21.391,-41.243
C01265=1014.750,231.623,-141.676,-24.397,21.391,-41.245
C01266=1014.748,231.374,-141.647,-24.397,21.392,-41.247
C01267=1014.746,231.126,-141.620,-24.396,21.392,-41.249
C01268=1014.743,230.877,-141.592,-24.396,21.392,-41.251
C01269=1014.741,230.628,-141.563,-24.396,21.391,-41.252
C01270=1014.738,230.386,-141.536,-24.396,21.392,-41.254
C01271=1014.736,230.142,-141.508,-24.395,21.392,-41.256
C01272=1014.733,229.900,-141.480,-24.395,21.392,-41.258
C01273=1014.730,229.657,-141.452,-24.395,21.392,-41.260
C01274=1014.729,229.414,-141.424,-24.395,21.392,-41.262
C01275=1014.726,229.171,-141.397,-24.394,21.392,-41.263
C01276=1014.724,228.928,-141.369,-24.394,21.392,-41.265
C01277=1014.722,228.686,-141.342,-24.394,21.393,-41.266
C01278=1014.719,228.437,-141.314,-24.394,21.393,-41.267
C01279=1014.717,228.188,-141.285,-24.394,21.393,-41.269
C01280=1014.714,227.940,-141.257,-24.393,21.394,-41.271
C01281=1014.712,227.691,-141.229,-24.393,21.393,-41.273
C01282=1014.710,227.443,-141.201,-24.393,21.393,-41.275
C01283=1014.708,227.195,-141.172,-24.393,21.393,-41.276
C01284=1014.705,226.947,-141.145,-24.392,21.394,-41.278
C01285=1014.702,226.698,-141.117,-24.392,21.394,-41.280
C01286=1014.700,226.449,-141.088,-24.392,21.393,-41.282
C01287=1014.698,226.201,-141.060,-24.391,21.393,-41.284
C01288=1014.696,225.953,-141.032,-24.391,21.394,-41.285
C01289=1014.693,225.704,-141.004,-24.391,21.395,-41.286
C01290=1014.691,225.456,-140.976,-24.391,21.395,-41.288
C01291=1014.689,225.208,-140.947,-24.391,21.394,-41.289
C01292=1014.687,224.959,-140.919,-24.390,21.394,-41.291
C01293=1014.684,224.711,-140.891,-24.390,21.395,-41.293
C01294=1014.682,224.463,-140.863,-24.390,21.395,-41.295
C01295=1014.679,224.214,-140.835,-24.390,21.395,-41.297
C01296=1014.677,223.966,-140.807,-24.389,21.394,-41.298
C01297=1014.675,223.717,-140.778,-24.389,21.395,-41.300
C01298=1014.672,223.475,-140.751,-24.389,21.395,-41.300
C01299=1014.670,223.232,-140.724,-24.389,21.396,-41.302
C01300=1014.669,222.989,-140.697,-24.389,21.396,-41.304
C01301=1014.666,222.746,-140.670,-24.388,21.395,-41.306
C01302=1014.663,222.503,-140.642,-24.388,21.395,-41.308
C01303=1014.662,222.260,-140.614,-24.388,21.396,-41.309
C01304=1014.659,222.018,-140.587,-24.388,21.397,-41.310
C01305=1014.657,221.775,-140.560,-24.388,21.396,-41.311
C01306=1014.655,221.526,-140.531,-24.387,21.396,-41.313
C01307=1014.653,221.278,-140.504,-24.387,21.396,-41.315
C01308=1014.651,221.030,-140.476,-24.387,21.397,-41.317
C01309=1014.648,220.781,-140.448,-24.386,21.396,-41.318
C01310=1014.646,220.533,-140.420,-24.386,21.396,-41.320
C01311=1014.644,220.285,-140.392,-24.386,21.397,-41.321
C01312=1014.642,220.036,-140.365,-24.386,21.397,-41.323
C01313=1014.640,219.787,-140.336,-24.386,21.397,-41.324
C01314=1014.638,219.540,-140.309,-24.385,21.397,-41.326
C01315=1014.636,219.290,-140.281,-24.385,21.397,-41.328
C01316=1014.633,219.042,-140.253,-24.385,21.397,-41.330
C01317=1014.632,218.794,-140.225,-24.385,21.397,-41.330
C01318=1014.629,218.545,-140.197,-24.385,21.397,-41.332
C01319=1014.627,218.297,-140.170,-24.384,21.398,-41.333
C01320=1014.625,218.049,-140.141,-24.384,21.398,-41.335
C01321=1014.622,217.800,-140.113,-24.384,21.397,-41.337
C01322=1014.621,217.551,-140.086,-24.384,21.397,-41.339
C01323=1014.618,217.303,-140.058,-24.384,21.398,-41.339
C01324=1014.617,217.055,-140.030,-24.383,21.399,-41.341
C01325=1014.614,216.806,-140.002,-24.383,21.398,-41.342
C01326=1014.612,216.563,-139.975,-24.383,21.398,-41.344
C01327=1014.611,216.321,-139.949,-24.383,21.398,-41.346
C01328=1014.609,216.078,-139.921,-24.383,21.398,-41.346
C01329=1014.606,215.836,-139.894,-24.382,21.399,-41.348
C01330=1014.604,215.593,-139.867,-24.382,21.399,-41.350
C01331=1014.603,215.350,-139.840,-24.382,21.399,-41.352
C01332=1014.600,215.107,-139.813,-24.382,21.398,-41.353
C01333=1014.598,214.865,-139.785,-24.382,21.399,-41.354
C01334=1014.597,214.616,-139.758,-24.381,21.400,-41.356
C01335=1014.594,214.368,-139.730,-24.381,21.399,-41.357
C01336=1014.592,214.119,-139.703,-24.381,21.399,-41.359
C01337=1014.591,213.871,-139.675,-24.381,21.400,-41.359
C01338=1014.589,213.623,-139.648,-24.381,21.400,-41.361
C01339=1014.586,213.374,-139.619,-24.380,21.400,-41.363
C01340=1014.584,213.125,-139.592,-24.380,21.400,-41.365
C01341=1014.583,212.877,-139.564,-24.380,21.400,-41.366
C01342=1014.581,212.629,-139.537,-24.380,21.400,-41.366
C01343=1014.578,212.381,-139.509,-24.380,21.400,-41.368
C01344=1014.577,212.132,-139.482,-24.379,21.400,-41.370
C01345=1014.575,211.883,-139.455,-24.379,21.400,-41.372
C01346=1014.573,211.634,-139.426,-24.379,21.401,-41.372
C01347=1014.571,211.386,-139.399,-24.379,21.401,-41.374
C01348=1014.569,211.138,-139.371,-24.378,21.400,-41.375
C01349=1014.567,210.889,-139.344,-24.378,21.400,-41.377
C01350=1014.566,210.640,-139.316,-24.378,21.401,-41.378
C01351=1014.563,210.393,-139.289,-24.378,21.401,-41.379
C01352=1014.561,210.144,-139.262,-24.378,21.401,-41.381
C01353=1014.560,209.895,-139.234,-24.377,21.401,-41.383
C01354=1014.558,209.653,-139.207,-24.377,21.401,-41.383
C01355=1014.556,209.411,-139.180,-24.377,21.401,-41.385
C01356=1014.555,209.167,-139.153,-24.377,21.402,-41.387
C01357=1014.552,208.925,-139.126,-24.377,21.401,-41.388
C01358=1014.551,208.682,-139.100,-24.377,21.402,-41.389
C01359=1014.548,208.440,-139.072,-24.376,21.402,-41.391
C01360=1014.547,208.197,-139.046,-24.376,21.401,-41.392
C01361=1014.545,207.955,-139.019,-24.376,21.402,-41.392
C01362=1014.543,207.706,-138.992,-24.376,21.402,-41.394
C01363=1014.542,207.457,-138.964,-24.376,21.402,-41.396
C01364=1014.540,207.209,-138.937,-24.375,21.402,-41.398
C01365=1014.538,206.961,-138.909,-24.375,21.402,-41.398
C01366=1014.536,206.712,-138.882,-24.375,21.402,-41.399
C01367=1014.534,206.464,-138.855,-24.375,21.402,-41.401
C01368=1014.533,206.215,-138.827,-24.375,21.402,-41.401
C01369=1014.530,205.967,-138.799,-24.375,21.403,-41.403
C01370=1014.529,205.718,-138.772,-24.374,21.403,-41.405
C01371=1014.527,205.470,-138.745,-24.374,21.402,-41.407
C01372=1014.525,205.221,-138.718,-24.374,21.403,-41.407
C01373=1014.524,204.972,-138.690,-24.374,21.403,-41.409
C01374=1014.522,204.724,-138.663,-24.373,21.403,-41.410
C01375=1014.521,204.476,-138.635,-24.374,21.404,-41.411
C01376=1014.519,204.228,-138.608,-24.373,21.403,-41.412
C01377=1014.517,203.979,-138.581,-24.373,21.403,-41.414
C01378=1014.515,203.730,-138.554,-24.373,21.404,-41.415
C01379=1014.514,203.482,-138.526,-24.373,21.403,-41.416
C01380=1014.509,202.266,-138.392,-24.425,21.378,-41.051
C01381=1014.509,201.879,-138.349,-24.424,21.378,-41.052
C01382=1014.510,201.530,-138.310,-24.424,21.378,-41.054
C01383=1014.510,201.178,-138.272,-24.424,21.378,-41.058
C01384=1014.511,200.771,-138.227,-24.423,21.379,-41.060
C01385=1014.511,200.544,-138.203,-24.423,21.378,-41.061
C01386=1014.512,200.315,-138.177,-24.423,21.378,-41.063
C01387=1014.512,200.091,-138.153,-24.423,21.378,-41.065
C01388=1014.513,199.879,-138.130,-24.423,21.378,-41.065
C01389=1014.514,199.478,-138.086,-24.422,21.379,-41.069
C01390=1014.515,199.089,-138.043,-24.422,21.379,-41.071
C01391=1014.516,198.691,-138.000,-24.421,21.379,-41.074
C01392=1014.516,198.290,-137.956,-24.421,21.379,-41.076
C01393=1014.518,197.889,-137.914,-24.421,21.380,-41.078
C01394=1014.519,197.487,-137.870,-24.420,21.380,-41.082
C01395=1014.520,197.087,-137.826,-24.420,21.380,-41.084
C01396=1014.520,196.686,-137.782,-24.419,21.380,-41.087
C01397=1014.522,196.284,-137.738,-24.419,21.380,-41.089
C01398=1014.523,195.883,-137.695,-24.419,21.381,-41.091
C01399=1014.523,195.482,-137.652,-24.418,21.380,-41.094
C01400=1014.525,195.080,-137.608,-24.418,21.381,-41.097
C01401=1014.525,194.680,-137.564,-24.418,21.381,-41.100
C01402=1014.527,194.279,-137.521,-24.417,21.381,-41.102
C01403=1014.527,193.878,-137.478,-24.417,21.381,-41.105
C01404=1014.529,193.476,-137.434,-24.417,21.382,-41.108
C01405=1014.530,193.075,-137.390,-24.416,21.382,-41.109
C01406=1014.531,192.675,-137.347,-24.416,21.382,-41.113
C01407=1014.532,192.273,-137.304,-24.415,21.382,-41.115
C01408=1014.533,191.872,-137.260,-24.415,21.382,-41.118
C01409=1014.534,191.471,-137.217,-24.415,21.382,-41.120
C01410=1014.535,191.070,-137.174,-24.414,21.382,-41.124
C01411=1014.536,190.669,-137.131,-24.414,21.383,-41.126
C01412=1014.537,190.267,-137.087,-24.414,21.383,-41.128
C01413=1014.539,189.867,-137.044,-24.413,21.383,-41.131
C01414=1014.540,189.466,-137.000,-24.413,21.383,-41.133
C01415=1014.541,189.065,-136.957,-24.412,21.384,-41.137
C01416=1014.542,188.664,-136.914,-24.412,21.384,-41.139
C01417=1014.543,188.262,-136.871,-24.412,21.384,-41.141
C01418=1014.545,187.861,-136.828,-24.411,21.384,-41.144
C01419=1014.546,187.460,-136.785,-24.411,21.385,-41.146
C01420=1014.547,187.060,-136.742,-24.411,21.384,-41.150
C01421=1014.548,186.658,-136.698,-24.410,21.384,-41.151
C01422=1014.549,186.258,-136.655,-24.410,21.384,-41.155
C01423=1014.550,185.856,-136.613,-24.410,21.385,-41.157
C01424=1014.552,185.455,-136.569,-24.409,21.385,-41.159
C01425=1014.553,185.055,-136.526,-24.409,21.385,-41.162
C01426=1014.554,184.653,-136.483,-24.409,21.386,-41.165
C01427=1014.556,184.253,-136.440,-24.408,21.386,-41.168
C01428=1014.557,183.851,-136.398,-24.408,21.386,-41.170
C01429=1014.558,183.451,-136.355,-24.407,21.386,-41.172
C01430=1014.559,183.050,-136.312,-24.407,21.386,-41.176
C01431=1014.561,182.649,-136.269,-24.407,21.387,-41.177
C01432=1014.562,182.248,-136.226,-24.406,21.386,-41.181
C01433=1014.563,181.847,-136.183,-24.406,21.387,-41.183
C01434=1014.564,181.447,-136.140,-24.405,21.387,-41.186
C01435=1014.566,181.046,-136.098,-24.405,21.387,-41.188
C01436=1014.567,180.644,-136.055,-24.405,21.387,-41.190
C01437=1014.568,180.244,-136.012,-24.404,21.388,-41.194
C01438=1014.570,179.843,-135.969,-24.404,21.388,-41.196
C01439=1014.571,179.442,-135.927,-24.403,21.388,-41.199
C01440=1014.573,179.041,-135.884,-24.403,21.388,-41.201
C01441=1014.574,178.641,-135.841,-24.403,21.388,-41.205
C01442=1014.576,178.240,-135.798,-24.402,21.388,-41.207
C01443=1014.577,177.839,-135.756,-24.402,21.389,-41.209
C01444=1014.578,177.438,-135.713,-24.402,21.389,-41.212
C01445=1014.580,177.037,-135.671,-24.401,21.389,-41.214
C01446=1014.581,176.636,-135.628,-24.401,21.389,-41.218
C01447=1014.582,176.236,-135.585,-24.401,21.389,-41.219
C01448=1014.585,175.835,-135.543,-24.400,21.390,-41.223
C01449=1014.585,175.435,-135.500,-24.400,21.390,-41.225
C01450=1014.587,175.034,-135.458,-24.400,21.390,-41.227
C01451=1014.588,174.633,-135.415,-24.399,21.390,-41.231
C01452=1014.590,174.232,-135.373,-24.399,21.391,-41.233
C01453=1014.591,173.832,-135.330,-24.398,21.390,-41.236
C01454=1014.593,173.431,-135.288,-24.398,21.390,-41.238
C01455=1014.593,173.030,-135.246,-24.397,21.391,-41.242
C01456=1014.595,172.629,-135.203,-24.397,21.391,-41.243
C01457=1014.597,172.230,-135.161,-24.397,21.391,-41.247
C01458=1014.599,171.828,-135.118,-24.396,21.392,-41.249
C01459=1014.599,171.428,-135.076,-24.396,21.392,-41.251
C01460=1014.602,171.028,-135.034,-24.396,21.392,-41.254
C01461=1014.603,170.627,-134.991,-24.395,21.392,-41.256
C01462=1014.605,170.226,-134.949,-24.395,21.392,-41.260
C01463=1014.605,169.825,-134.907,-24.395,21.392,-41.262
C01464=1014.607,169.426,-134.865,-24.394,21.392,-41.265
C01465=1014.609,169.024,-134.823,-24.394,21.393,-41.267
C01466=1014.610,168.625,-134.781,-24.393,21.393,-41.271
C01467=1014.612,168.224,-134.738,-24.393,21.393,-41.273
C01468=1014.614,167.824,-134.696,-24.393,21.394,-41.275
C01469=1014.615,167.423,-134.654,-24.392,21.394,-41.278
C01470=1014.617,167.023,-134.612,-24.392,21.394,-41.280
C01471=1014.618,166.623,-134.570,-24.391,21.393,-41.284
C01472=1014.620,166.222,-134.528,-24.391,21.395,-41.286
C01473=1014.622,165.821,-134.486,-24.391,21.394,-41.289
C01474=1014.623,165.422,-134.444,-24.390,21.394,-41.291
C01475=1014.624,165.020,-134.402,-24.390,21.395,-41.295
C01476=1014.626,164.621,-134.360,-24.390,21.395,-41.297
C01477=1014.628,164.221,-134.318,-24.389,21.395,-41.300
C01478=1014.629,163.834,-134.277,-24.389,21.395,-41.302
C01479=1014.630,163.644,-134.258,-24.389,21.395,-41.304
C01480=1014.631,163.233,-134.214,-24.388,21.396,-41.306
C01481=1014.632,162.997,-134.189,-24.388,21.395,-41.308
C01482=1014.633,162.743,-134.163,-24.388,21.396,-41.309
C01483=1014.635,162.480,-134.136,-24.388,21.396,-41.311
C01484=1014.635,162.211,-134.107,-24.387,21.396,-41.313
C01485=1014.637,161.940,-134.080,-24.387,21.396,-41.315
C01486=1014.638,161.671,-134.051,-24.387,21.397,-41.317
C01487=1014.639,161.409,-134.023,-24.387,21.397,-41.319
C01488=1014.640,161.157,-133.997,-24.386,21.396,-41.320
C01489=1014.641,160.920,-133.973,-24.386,21.396,-41.322
C01490=1014.641,160.696,-133.949,-24.386,21.397,-41.324
C01491=1014.643,160.482,-133.927,-24.386,21.397,-41.325
C01492=1014.644,160.077,-133.885,-24.385,21.397,-41.328
C01493=1014.647,159.680,-133.844,-24.385,21.397,-41.330
C01494=1014.655,159.281,-133.806,-24.384,21.398,-41.333
C01495=1014.663,158.880,-133.769,-24.384,21.398,-41.335
C01496=1014.672,158.479,-133.732,-24.384,21.397,-41.339
C01497=1014.680,158.077,-133.693,-24.383,21.399,-41.341
C01498=1014.689,157.674,-133.655,-24.383,21.398,-41.344
C01499=1014.697,157.271,-133.617,-24.383,21.398,-41.346
C01500=1014.704,156.867,-133.579,-24.382,21.399,-41.350
C01501=1014.713,156.462,-133.542,-24.382,21.399,-41.352
C01502=1014.721,156.057,-133.503,-24.381,21.399,-41.355
C01503=1014.729,155.650,-133.465,-24.381,21.400,-41.358
C01504=1014.737,155.242,-133.426,-24.381,21.399,-41.361
C01505=1014.745,154.833,-133.388,-24.380,21.400,-41.363
C01506=1014.753,154.425,-133.349,-24.380,21.400,-41.366
C01507=1014.761,154.015,-133.311,-24.380,21.400,-41.368
C01508=1014.770,153.604,-133.272,-24.379,21.401,-41.372
C01509=1014.777,153.193,-133.234,-24.378,21.400,-41.375
C01510=1014.785,152.782,-133.195,-24.378,21.400,-41.377
C01511=1014.794,152.369,-133.155,-24.378,21.401,-41.381
C01512=1014.802,151.957,-133.116,-24.377,21.401,-41.383
C01513=1014.809,151.544,-133.078,-24.377,21.402,-41.387
C01514=1014.818,151.131,-133.039,-24.377,21.402,-41.389
C01515=1014.825,150.717,-133.000,-24.376,21.401,-41.392
C01516=1014.833,150.304,-132.961,-24.376,21.402,-41.394
C01517=1014.841,149.890,-132.922,-24.375,21.402,-41.398
C01518=1014.849,149.476,-132.884,-24.375,21.402,-41.401
C01519=1014.857,149.062,-132.844,-24.375,21.403,-41.403
C01520=1014.865,148.648,-132.805,-24.374,21.403,-41.407
C01521=1014.872,148.234,-132.766,-24.374,21.403,-41.409
C01522=1014.880,147.820,-132.727,-24.373,21.403,-41.412
C01523=1014.887,147.425,-132.690,-24.373,21.403,-41.416
C01524=1014.894,147.031,-132.653,-24.372,21.404,-41.418
C01525=1014.903,146.580,-132.610,-24.372,21.404,-41.422
C01526=1014.910,146.167,-132.571,-24.372,21.404,-41.424
C01527=1014.918,145.753,-132.533,-24.371,21.405,-41.427
C01528=1014.925,145.341,-132.494,-24.371,21.404,-41.431
C01529=1014.933,144.929,-132.455,-24.370,21.405,-41.432
C01530=1014.941,144.518,-132.417,-24.370,21.405,-41.436
C01531=1014.948,144.108,-132.378,-24.370,21.405,-41.438
C01532=1014.955,143.697,-132.339,-24.369,21.406,-41.442
C01533=1014.963,143.288,-132.301,-24.369,21.405,-41.445
C01534=1014.970,142.879,-132.262,-24.368,21.406,-41.448
C01535=1014.977,142.471,-132.224,-24.368,21.406,-41.451
C01536=1014.985,142.064,-132.185,-24.368,21.406,-41.453
C01537=1014.991,141.658,-132.147,-24.367,21.407,-41.457
C01538=1014.999,141.253,-132.109,-24.366,21.406,-41.460
C01539=1015.006,140.848,-132.070,-24.366,21.407,-41.462
C01540=1015.013,140.431,-132.031,-24.366,21.408,-41.466
C01541=1015.018,140.195,-132.009,-24.366,21.408,-41.468
C01542=1015.022,139.936,-131.984,-24.365,21.408,-41.470
C01543=1015.026,139.659,-131.958,-24.365,21.408,-41.471
C01544=1015.032,139.372,-131.931,-24.365,21.408,-41.473
C01545=1015.036,139.084,-131.905,-24.364,21.408,-41.475
C01546=1015.042,138.807,-131.879,-24.364,21.407,-41.476
C01547=1015.046,138.547,-131.854,-24.364,21.408,-41.478
C01548=1015.050,138.309,-131.832,-24.364,21.408,-41.480
C01549=1015.054,138.093,-131.810,-24.363,21.408,-41.482
C01550=1015.058,137.887,-131.792,-24.363,21.408,-41.484
C01551=1015.064,137.486,-131.754,-24.363,21.408,-41.486
C01552=1015.070,137.115,-131.719,-24.363,21.410,-41.488
C01553=1015.076,136.780,-131.688,-24.362,21.409,-41.491
C01554=1015.082,136.463,-131.658,-24.361,21.409,-41.495
C01555=1015.087,136.146,-131.627,-24.361,21.410,-41.497
C01556=1015.092,135.806,-131.596,-24.361,21.409,-41.500
C01557=1015.099,135.435,-131.561,-24.360,21.410,-41.502
C01558=1015.106,135.040,-131.523,-24.360,21.411,-41.505
C01559=1015.112,134.640,-131.486,-24.360,21.410,-41.508
C01560=1015.119,134.242,-131.448,-24.359,21.411,-41.510
C01561=1015.125,133.844,-131.411,-24.359,21.411,-41.514
C01562=1015.132,133.445,-131.374,-24.358,21.411,-41.517
C01563=1015.138,133.046,-131.336,-24.358,21.412,-41.519
C01564=1015.145,132.648,-131.298,-24.358,21.411,-41.523
C01565=1015.151,132.249,-131.261,-24.357,21.412,-41.525
C01566=1015.158,131.850,-131.223,-24.357,21.412,-41.528
C01567=1015.164,131.452,-131.186,-24.356,21.412,-41.532
C01568=1015.171,131.053,-131.148,-24.356,21.413,-41.534
C01569=1015.177,130.655,-131.112,-24.356,21.413,-41.538
C01570=1015.183,130.256,-131.074,-24.355,21.413,-41.541
C01571=1015.189,129.858,-131.036,-24.355,21.413,-41.543
C01572=1015.196,129.460,-130.998,-24.354,21.413,-41.547
C01573=1015.202,129.061,-130.960,-24.354,21.413,-41.550
C01574=1015.209,128.662,-130.924,-24.354,21.414,-41.552
C01575=1015.215,128.264,-130.886,-24.353,21.414,-41.555
C01576=1015.221,127.865,-130.849,-24.353,21.415,-41.558
C01577=1015.228,127.467,-130.811,-24.352,21.414,-41.561
C01578=1015.233,127.068,-130.774,-24.352,21.415,-41.565
C01579=1015.240,126.669,-130.737,-24.351,21.415,-41.567
C01580=1015.246,126.271,-130.699,-24.351,21.415,-41.571
C01581=1015.252,125.873,-130.662,-24.350,21.415,-41.574
C01582=1015.258,125.474,-130.624,-24.350,21.416,-41.576
C01583=1015.264,125.076,-130.587,-24.350,21.416,-41.580
C01584=1015.270,124.677,-130.549,-24.349,21.416,-41.583
C01585=1015.276,124.279,-130.511,-24.349,21.416,-41.585
C01586=1015.282,123.880,-130.474,-24.348,21.417,-41.589
C01587=1015.289,123.482,-130.437,-24.348,21.416,-41.592
C01588=1015.294,123.083,-130.400,-24.348,21.418,-41.595
C01589=1015.300,122.684,-130.362,-24.347,21.417,-41.598
C01590=1015.306,122.286,-130.325,-24.347,21.418,-41.602
C01591=1015.313,121.888,-130.287,-24.346,21.417,-41.605
C01592=1015.318,121.490,-130.250,-24.346,21.418,-41.607
C01593=1015.324,121.091,-130.212,-24.345,21.418,-41.611
C01594=1015.330,120.692,-130.175,-24.345,21.418,-41.614
C01595=1015.336,120.295,-130.138,-24.345,21.419,-41.617
C01596=1015.342,119.895,-130.100,-24.344,21.419,-41.620
C01597=1015.348,119.498,-130.064,-24.343,21.419,-41.624
C01598=1015.355,119.098,-130.026,-24.343,21.420,-41.626
C01599=1015.361,118.700,-129.989,-24.343,21.420,-41.629
C01600=1015.366,118.302,-129.952,-24.342,21.420,-41.633
C01601=1015.373,117.903,-129.915,-24.342,21.420,-41.637
C01602=1015.379,117.505,-129.878,-24.341,21.420,-41.638
C01603=1015.386,117.107,-129.841,-24.341,21.421,-41.642
C01604=1015.391,116.708,-129.804,-24.340,21.420,-41.646
C01605=1015.397,116.310,-129.767,-24.340,21.421,-41.649
C01606=1015.404,115.911,-129.730,-24.340,21.422,-41.652
C01607=1015.410,115.513,-129.693,-24.339,21.422,-41.655
C01608=1015.415,115.115,-129.656,-24.339,21.422,-41.659
C01609=1015.421,114.716,-129.619,-24.338,21.422,-41.662
C01610=1015.428,114.318,-129.582,-24.338,21.423,-41.664
C01611=1015.433,113.919,-129.544,-24.337,21.422,-41.668
C01612=1015.439,113.520,-129.508,-24.337,21.423,-41.671
C01613=1015.445,113.122,-129.471,-24.336,21.423,-41.675
C01614=1015.450,112.724,-129.433,-24.336,21.423,-41.677
C01615=1015.457,112.325,-129.396,-24.335,21.424,-41.681
C01616=1015.463,111.927,-129.359,-24.335,21.423,-41.684
C01617=1015.468,111.528,-129.322,-24.334,21.424,-41.688
C01618=1015.474,111.129,-129.286,-24.334,21.425,-41.690
C01619=1015.480,110.731,-129.248,-24.334,21.425,-41.694
C01620=1015.486,110.333,-129.211,-24.333,21.425,-41.697
C01621=1015.491,109.934,-129.175,-24.333,21.425,-41.701
C01622=1015.497,109.536,-129.137,-24.332,21.426,-41.703
C01623=1015.502,109.137,-129.100,-24.332,21.426,-41.707
C01624=1015.508,108.738,-129.064,-24.331,21.426,-41.710
C01625=1015.514,108.341,-129.027,-24.331,21.426,-41.714
C01626=1015.519,107.942,-128.989,-24.330,21.426,-41.717
C01627=1015.525,107.543,-128.953,-24.330,21.427,-41.719
C01628=1015.531,107.145,-128.915,-24.330,21.427,-41.723
C01629=1015.536,106.746,-128.878,-24.329,21.427,-41.727
C01630=1015.542,106.347,-128.842,-24.328,21.427,-41.730
C01631=1015.547,105.949,-128.804,-24.328,21.428,-41.734
C01632=1015.553,105.550,-128.767,-24.328,21.428,-41.736
C01633=1015.558,105.151,-128.730,-24.327,21.429,-41.740
C01634=1015.563,104.753,-128.694,-24.327,21.429,-41.743
C01635=1015.569,104.354,-128.657,-24.326,21.429,-41.747
C01636=1015.574,103.956,-128.620,-24.326,21.429,-41.751
C01637=1015.580,103.557,-128.583,-24.325,21.430,-41.754
C01638=1015.585,103.158,-128.546,-24.325,21.430,-41.756
C01639=1015.590,102.760,-128.509,-24.324,21.430,-41.760
C01640=1015.596,102.362,-128.472,-24.324,21.430,-41.763
C01641=1015.601,101.963,-128.435,-24.323,21.430,-41.767
C01642=1015.607,101.564,-128.398,-24.323,21.431,-41.771
C01643=1015.612,101.165,-128.362,-24.322,21.431,-41.775
C01644=1015.617,100.766,-128.325,-24.322,21.431,-41.778
C01645=1015.622,100.368,-128.287,-24.322,21.432,-41.780
C01646=1015.627,99.969,-128.251,-24.321,21.432,-41.784
C01647=1015.632,99.571,-128.214,-24.320,21.432,-41.787
C01648=1015.638,99.171,-128.177,-24.320,21.432,-41.791
C01649=1015.642,98.773,-128.140,-24.319,21.433,-41.795
C01650=1015.648,98.374,-128.104,-24.319,21.432,-41.798
C01651=1015.653,97.976,-128.067,-24.318,21.433,-41.802
C01652=1015.658,97.576,-128.029,-24.318,21.433,-41.806
C01653=1015.663,97.177,-127.993,-24.318,21.434,-41.808
C01654=1015.668,96.779,-127.956,-24.317,21.434,-41.811
C01655=1015.673,96.380,-127.919,-24.317,21.435,-41.815
C01656=1015.678,95.981,-127.882,-24.316,21.435,-41.819
C01657=1015.683,95.582,-127.846,-24.316,21.435,-41.822
C01658=1015.688,95.184,-127.809,-24.315,21.435,-41.826
C01659=1015.693,94.784,-127.772,-24.315,21.436,-41.830
C01660=1015.697,94.386,-127.735,-24.314,21.435,-41.833
C01661=1015.703,93.986,-127.698,-24.313,21.436,-41.837
C01662=1015.707,93.588,-127.662,-24.313,21.436,-41.841
C01663=1015.712,93.188,-127.625,-24.312,21.437,-41.844
C01664=1015.717,92.790,-127.588,-24.312,21.437,-41.846
C01665=1015.722,92.390,-127.552,-24.312,21.437,-41.850
C01666=1015.727,91.991,-127.515,-24.311,21.438,-41.854
C01667=1015.731,91.593,-127.478,-24.311,21.438,-41.857
C01668=1015.737,91.193,-127.441,-24.310,21.438,-41.861
C01669=1015.741,90.794,-127.404,-24.310,21.438,-41.865
C01670=1015.746,90.395,-127.368,-24.309,21.439,-41.868
C01671=1015.751,89.995,-127.331,-24.309,21.439,-41.872
C01672=1015.755,89.597,-127.294,-24.308,21.439,-41.875
C01673=1015.760,89.205,-127.258,-24.308,21.439,-41.879
C01674=1015.764,88.818,-127.222,-24.307,21.440,-41.883
C01675=1015.769,88.436,-127.188,-24.307,21.440,-41.887
C01676=1015.773,88.053,-127.152,-24.306,21.440,-41.890
C01677=1015.778,87.664,-127.116,-24.305,21.440,-41.894
C01678=1015.782,87.267,-127.080,-24.305,21.441,-41.898
C01679=1015.787,86.865,-127.043,-24.304,21.441,-41.901
C01680=1015.791,86.459,-127.006,-24.304,21.442,-41.905
C01681=1015.796,86.052,-126.968,-24.303,21.441,-41.908
C01682=1015.800,85.643,-126.931,-24.303,21.442,-41.912
C01683=1015.805,85.232,-126.893,-24.302,21.442,-41.916
C01684=1015.810,84.820,-126.855,-24.302,21.443,-41.920
C01685=1015.814,84.406,-126.817,-24.301,21.443,-41.923
C01686=1015.819,83.990,-126.779,-24.301,21.443,-41.927
C01687=1015.823,83.572,-126.740,-24.300,21.444,-41.931
C01688=1015.828,83.154,-126.702,-24.300,21.444,-41.935
C01689=1015.833,82.734,-126.664,-24.299,21.444,-41.938
C01690=1015.837,82.312,-126.626,-24.299,21.444,-41.942
C01691=1015.839,82.101,-126.606,-24.299,21.445,-41.944
C01692=1015.841,81.889,-126.587,-24.298,21.444,-41.947
C01693=1015.844,81.678,-126.567,-24.298,21.445,-41.949
C01694=1015.846,81.466,-126.548,-24.298,21.445,-41.951
C01695=1015.848,81.254,-126.528,-24.297,21.445,-41.953
C01696=1015.850,81.041,-126.509,-24.297,21.445,-41.955
C01697=1015.852,80.829,-126.489,-24.297,21.445,-41.956
C01698=1015.855,80.616,-126.470,-24.297,21.446,-41.958
C01699=1015.857,80.403,-126.450,-24.296,21.446,-41.960
C01700=1015.860,80.190,-126.431,-24.296,21.446,-41.962
C01701=1015.862,79.978,-126.412,-24.296,21.446,-41.964
C01702=1015.864,79.768,-126.393,-24.296,21.447,-41.966
C01703=1015.868,79.354,-126.354,-24.295,21.447,-41.970
C01704=1015.872,78.948,-126.317,-24.294,21.447,-41.973
C01705=1015.877,78.551,-126.281,-24.294,21.447,-41.977
C01706=1015.881,78.160,-126.245,-24.293,21.448,-41.980
C01707=1015.885,77.774,-126.210,-24.293,21.447,-41.986
C01708=1015.888,77.388,-126.175,-24.292,21.448,-41.989
C01709=1015.893,76.999,-126.139,-24.292,21.449,-41.994
C01710=1015.897,76.605,-126.104,-24.291,21.449,-41.997
C01711=1015.901,76.203,-126.066,-24.291,21.449,-42.001
C01712=1015.905,75.791,-126.029,-24.290,21.450,-42.004
C01713=1015.909,75.372,-125.990,-24.290,21.450,-42.008
C01714=1015.911,75.159,-125.971,-24.289,21.451,-42.010
C01715=1015.913,74.946,-125.952,-24.289,21.451,-42.012
C01716=1015.916,74.732,-125.933,-24.289,21.450,-42.015
C01717=1015.917,74.519,-125.913,-24.288,21.451,-42.017
C01718=1015.920,74.306,-125.894,-24.288,21.451,-42.019
C01719=1015.922,74.093,-125.874,-24.288,21.451,-42.021
C01720=1015.924,73.881,-125.855,-24.288,21.451,-42.023
C01721=1015.926,73.670,-125.835,-24.287,21.452,-42.025
C01722=1015.930,73.249,-125.798,-24.287,21.452,-42.028
C01723=1015.934,72.831,-125.759,-24.286,21.452,-42.034
C01724=1015.938,72.416,-125.722,-24.285,21.452,-42.037
C01725=1015.942,72.002,-125.684,-24.285,21.453,-42.041
C01726=1015.946,71.591,-125.647,-24.285,21.453,-42.045
C01727=1015.949,71.179,-125.609,-24.284,21.454,-42.049
C01728=1015.954,70.768,-125.572,-24.283,21.453,-42.054
C01729=1015.958,70.358,-125.535,-24.283,21.454,-42.058
C01730=1015.961,69.945,-125.497,-24.282,21.454,-42.061
C01731=1015.966,69.535,-125.460,-24.282,21.455,-42.065
C01732=1015.969,69.125,-125.423,-24.281,21.455,-42.069
C01733=1015.973,68.716,-125.386,-24.280,21.455,-42.074
C01734=1015.977,68.309,-125.348,-24.280,21.456,-42.078
C01735=1015.980,67.903,-125.312,-24.279,21.456,-42.082
C01736=1015.984,67.498,-125.274,-24.279,21.457,-42.085
C01737=1015.988,67.095,-125.238,-24.278,21.457,-42.089
C01738=1015.991,66.692,-125.202,-24.278,21.457,-42.094
C01739=1015.995,66.291,-125.166,-24.277,21.457,-42.098
C01740=1015.998,65.894,-125.130,-24.277,21.458,-42.102
C01741=1016.002,65.486,-125.092,-24.276,21.458,-42.106
C01742=1016.004,65.272,-125.073,-24.276,21.459,-42.108
C01743=1016.006,65.052,-125.054,-24.275,21.458,-42.111
C01744=1016.008,64.822,-125.033,-24.275,21.458,-42.113
C01745=1016.009,64.586,-125.011,-24.275,21.459,-42.115
C01746=1016.012,64.350,-124.990,-24.274,21.459,-42.116
C01747=1016.014,64.121,-124.969,-24.274,21.459,-42.120
C01748=1016.016,63.903,-124.949,-24.274,21.460,-42.122
C01749=1016.018,63.696,-124.930,-24.274,21.460,-42.124
C01750=1016.020,63.479,-124.911,-24.273,21.459,-42.127
C01751=1016.022,63.228,-124.888,-24.273,21.460,-42.129
C01752=1016.024,62.962,-124.865,-24.272,21.460,-42.131
C01753=1016.026,62.708,-124.841,-24.272,21.460,-42.133
C01754=1016.030,62.289,-124.803,-24.271,21.461,-42.139
C01755=1016.033,61.888,-124.768,-24.271,21.461,-42.142
C01756=1016.037,61.488,-124.731,-24.270,21.462,-42.146
C01757=1016.039,61.088,-124.695,-24.270,21.462,-42.150
C01758=1016.043,60.688,-124.659,-24.269,21.462,-42.155
C01759=1016.046,60.287,-124.623,-24.269,21.463,-42.159
C01760=1016.050,59.887,-124.586,-24.268,21.463,-42.163
C01761=1016.053,59.487,-124.550,-24.268,21.464,-42.166
C01762=1016.056,59.087,-124.515,-24.267,21.463,-42.172
C01763=1016.059,58.687,-124.479,-24.266,21.464,-42.175
C01764=1016.062,58.287,-124.443,-24.266,21.464,-42.179
C01765=1016.066,57.886,-124.407,-24.265,21.465,-42.183
C01766=1016.069,57.486,-124.371,-24.264,21.465,-42.188
C01767=1016.073,57.087,-124.334,-24.264,21.465,-42.192
C01768=1016.075,56.685,-124.299,-24.264,21.466,-42.196
C01769=1016.078,56.286,-124.263,-24.263,21.465,-42.201
C01770=1016.081,55.886,-124.226,-24.262,21.467,-42.205
C01771=1016.085,55.485,-124.191,-24.262,21.467,-42.209
C01772=1016.088,55.085,-124.155,-24.261,21.468,-42.212
C01773=1016.091,54.686,-124.119,-24.260,21.468,-42.218
C01774=1016.094,54.285,-124.083,-24.260,21.468,-42.221
C01775=1016.097,53.884,-124.047,-24.259,21.468,-42.225
C01776=1016.100,53.485,-124.011,-24.259,21.468,-42.230
C01777=1016.103,53.084,-123.975,-24.258,21.469,-42.234
C01778=1016.106,52.685,-123.940,-24.258,21.469,-42.238
C01779=1016.109,52.285,-123.904,-24.257,21.469,-42.243
C01780=1016.111,51.884,-123.868,-24.256,21.470,-42.247
C01781=1016.114,51.484,-123.832,-24.256,21.471,-42.251
C01782=1016.118,51.084,-123.796,-24.255,21.471,-42.255
C01783=1016.120,50.684,-123.761,-24.255,21.471,-42.260
C01784=1016.123,50.284,-123.725,-24.254,21.472,-42.264
C01785=1016.126,49.883,-123.689,-24.254,21.472,-42.268
C01786=1016.128,49.483,-123.653,-24.253,21.472,-42.273
C01787=1016.131,49.083,-123.617,-24.252,21.473,-42.277
